LIN {X 0,Y 354.919,Z 337.275,A -85,B 0,C 180,E1 -13602.581,E2 -13602.581} C_VEL
LIN {X 0,Y 354.887,Z 337.28,A -85,B 0,C 180,E1 -13606.096,E2 -13606.096} C_VEL
LIN {X 0,Y 354.904,Z 337.277,A -85,B 0,C 180,E1 -13608.472,E2 -13608.472} C_VEL
LIN {X 0,Y 354.833,Z 337.288,A -85,B 0,C 180,E1 -13612.107,E2 -13612.107} C_VEL
LIN {X 0,Y 354.897,Z 337.277,A -85,B 0,C 180,E1 -13615.828,E2 -13615.828} C_VEL
LIN {X 0,Y 354.816,Z 337.287,A -85,B 0,C 180,E1 -13619.682,E2 -13619.682} C_VEL
LIN {X 0,Y 354.805,Z 337.288,A -85,B 0,C 180,E1 -13623.703,E2 -13623.703} C_VEL
LIN {X 0,Y 354.798,Z 337.29,A -85,B 0,C 180,E1 -13626.46,E2 -13626.46} C_VEL
LIN {X 0,Y 354.823,Z 337.285,A -85,B 0,C 180,E1 -13629.424,E2 -13629.424} C_VEL
LIN {X 0,Y 354.786,Z 337.289,A -85,B 0,C 180,E1 -13632.695,E2 -13632.695} C_VEL
LIN {X 0,Y 354.114,Z 337.376,A -85,B 0,C 180,E1 -13633.641,E2 -13633.641} C_VEL
LIN {X 0,Y 351.229,Z 337.732,A -85,B 0,C 180,E1 -13635.178,E2 -13635.178} C_VEL
LIN {X 0,Y 348.801,Z 338.036,A -85,B 0,C 180,E1 -13636.423,E2 -13636.423} C_VEL
LIN {X 0,Y 347.786,Z 338.161,A -85,B 0,C 180,E1 -13637.387,E2 -13637.387} C_VEL
LIN {X 0,Y 347.718,Z 338.169,A -85,B 0,C 180,E1 -13637.713,E2 -13637.713} C_VEL
LIN {X 0,Y 347.752,Z 338.165,A -85,B 0,C 180,E1 -13641.208,E2 -13641.208} C_VEL
LIN {X 0,Y 347.789,Z 338.164,A -85,B 0,C 180,E1 -13644.126,E2 -13644.126} C_VEL
LIN {X 0,Y 347.74,Z 338.17,A -85,B 0,C 180,E1 -13648.087,E2 -13648.087} C_VEL
LIN {X 0,Y 347.866,Z 338.151,A -85,B 0,C 180,E1 -13651.134,E2 -13651.134} C_VEL
LIN {X 0,Y 354.099,Z 357.245,A -85,B 0,C 180,E1 -13651.928,E2 -13651.928} C_VEL
LIN {X 0,Y 352.575,Z 425.531,A -85,B 0,C 180,E1 -13653.715,E2 -13653.715} C_VEL
LIN {X 0,Y 352.322,Z 438.618,A -85,B 0,C 180,E1 -13654.288,E2 -13654.288} C_VEL
LIN {X 0,Y 351.875,Z 452.101,A -85,B 0,C 180,E1 -13655.123,E2 -13655.123} C_VEL
LIN {X 0,Y 351.307,Z 464.045,A -85,B 0,C 180,E1 -13656.103,E2 -13656.103} C_VEL
LIN {X 0,Y 350.651,Z 475.904,A -85,B 0,C 180,E1 -13657.337,E2 -13657.337} C_VEL
LIN {X 0,Y 349.975,Z 486.089,A -85,B 0,C 180,E1 -13658.656,E2 -13658.656} C_VEL
LIN {X 0,Y 349.313,Z 494.652,A -85,B 0,C 180,E1 -13660,E2 -13660} C_VEL
LIN {X 0,Y 348.778,Z 502.203,A -85,B 0,C 180,E1 -13661.422,E2 -13661.422} C_VEL
LIN {X 0,Y 348.23,Z 510.285,A -85,B 0,C 180,E1 -13663.287,E2 -13663.287} C_VEL
LIN {X 0,Y 347.925,Z 515.474,A -85,B 0,C 180,E1 -13664.776,E2 -13664.776} C_VEL
LIN {X 0,Y 347.638,Z 520.436,A -85,B 0,C 180,E1 -13666.557,E2 -13666.557} C_VEL
LIN {X 0,Y 347.438,Z 524.191,A -85,B 0,C 180,E1 -13668.33,E2 -13668.33} C_VEL
LIN {X 0,Y 347.413,Z 526.086,A -85,B 0,C 180,E1 -13669.51,E2 -13669.51} C_VEL
LIN {X 0,Y 347.453,Z 527.538,A -85,B 0,C 180,E1 -13670.688,E2 -13670.688} C_VEL
LIN {X 0,Y 347.593,Z 528.701,A -85,B 0,C 180,E1 -13672.198,E2 -13672.198} C_VEL
LIN {X 0,Y 347.785,Z 529.183,A -85,B 0,C 180,E1 -13674.202,E2 -13674.202} C_VEL
LIN {X 0,Y 347.848,Z 528.865,A -85,B 0,C 180,E1 -13675.365,E2 -13675.365} C_VEL
LIN {X 0,Y 348.18,Z 528.105,A -85,B 0,C 180,E1 -13676.529,E2 -13676.529} C_VEL
LIN {X 0,Y 348.507,Z 526.945,A -85,B 0,C 180,E1 -13677.689,E2 -13677.689} C_VEL
LIN {X 0,Y 349.141,Z 524.323,A -85,B 0,C 180,E1 -13679.424,E2 -13679.424} C_VEL
LIN {X 0,Y 349.883,Z 520.636,A -85,B 0,C 180,E1 -13681.152,E2 -13681.152} C_VEL
LIN {X 0,Y 350.847,Z 515.743,A -85,B 0,C 180,E1 -13682.871,E2 -13682.871} C_VEL
LIN {X 0,Y 351.922,Z 509.602,A -85,B 0,C 180,E1 -13684.582,E2 -13684.582} C_VEL
LIN {X 0,Y 353.246,Z 501.914,A -85,B 0,C 180,E1 -13686.283,E2 -13686.283} C_VEL
LIN {X 0,Y 354.34,Z 494.044,A -85,B 0,C 180,E1 -13687.694,E2 -13687.694} C_VEL
LIN {X 0,Y 355.681,Z 484.348,A -85,B 0,C 180,E1 -13689.096,E2 -13689.096} C_VEL
LIN {X 0,Y 356.808,Z 473.673,A -85,B 0,C 180,E1 -13690.355,E2 -13690.355} C_VEL
LIN {X 0,Y 357.981,Z 461.641,A -85,B 0,C 180,E1 -13691.466,E2 -13691.466} C_VEL
LIN {X 0,Y 358.844,Z 448.971,A -85,B 0,C 180,E1 -13692.37,E2 -13692.37} C_VEL
LIN {X 0,Y 359.418,Z 435.559,A -85,B 0,C 180,E1 -13693.068,E2 -13693.068} C_VEL
LIN {X 0,Y 359.955,Z 415.445,A -85,B 0,C 180,E1 -13693.729,E2 -13693.729} C_VEL
LIN {X 0,Y 362.512,Z 365.478,A -85,B 0,C 180,E1 -13695.192,E2 -13695.192} C_VEL
LIN {X 0,Y 357.377,Z 355.182,A -85,B 0,C 180,E1 -13696.181,E2 -13696.181} C_VEL
LIN {X 0,Y 352.177,Z 346.136,A -85,B 0,C 180,E1 -13697.226,E2 -13697.226} C_VEL
LIN {X 0,Y 349.985,Z 342.457,A -85,B 0,C 180,E1 -13697.684,E2 -13697.684} C_VEL
LIN {X 0,Y 348.202,Z 339.745,A -85,B 0,C 180,E1 -13698.061,E2 -13698.061} C_VEL
LIN {X 0,Y 347.81,Z 338.162,A -85,B 0,C 180,E1 -13698.193,E2 -13698.193} C_VEL
LIN {X 0,Y 347.767,Z 338.171,A -85,B 0,C 180,E1 -13701.624,E2 -13701.624} C_VEL
LIN {X 0,Y 347.742,Z 338.171,A -85,B 0,C 180,E1 -13705.114,E2 -13705.114} C_VEL
LIN {X 0,Y 347.732,Z 338.171,A -85,B 0,C 180,E1 -13707.701,E2 -13707.701} C_VEL
LIN {X 0,Y 347.742,Z 338.169,A -85,B 0,C 180,E1 -13710.349,E2 -13710.349} C_VEL
LIN {X 0,Y 347.752,Z 338.167,A -85,B 0,C 180,E1 -13714.044,E2 -13714.044} C_VEL
LIN {X 0,Y 347.758,Z 338.163,A -85,B 0,C 180,E1 -13717.322,E2 -13717.322} C_VEL
LIN {X 0,Y 347.7,Z 338.171,A -85,B 0,C 180,E1 -13720.302,E2 -13720.302} C_VEL
LIN {X 0,Y 347.725,Z 338.169,A -85,B 0,C 180,E1 -13723.409,E2 -13723.409} C_VEL
LIN {X 0,Y 347.728,Z 338.171,A -85,B 0,C 180,E1 -13726.687,E2 -13726.687} C_VEL
LIN {X 0,Y 347.704,Z 338.174,A -85,B 0,C 180,E1 -13730.182,E2 -13730.182} C_VEL
LIN {X 0,Y 347.76,Z 338.167,A -85,B 0,C 180,E1 -13732.678,E2 -13732.678} C_VEL
LIN {X 0,Y 347.845,Z 338.187,A -85,B 0,C 180,E1 -13736.04,E2 -13736.04} C_VEL
LIN {X 0,Y 351.883,Z 357.108,A -85,B 0,C 180,E1 -13740.045,E2 -13740.045} C_VEL
LIN {X 0,Y 352.906,Z 362.731,A -85,B 0,C 180,E1 -13741.194,E2 -13741.194} C_VEL
LIN {X 0,Y 351.557,Z 377.008,A -85,B 0,C 180,E1 -13743.868,E2 -13743.868} C_VEL
LIN {X 0,Y 354.305,Z 396.014,A -85,B 0,C 180,E1 -13744.981,E2 -13744.981} C_VEL
LIN {X 0,Y 357.252,Z 419.557,A -85,B 0,C 180,E1 -13746.175,E2 -13746.175} C_VEL
LIN {X 0,Y 358.896,Z 440.791,A -85,B 0,C 180,E1 -13747.091,E2 -13747.091} C_VEL
LIN {X 0,Y 359.227,Z 450.079,A -85,B 0,C 180,E1 -13747.438,E2 -13747.438} C_VEL
LIN {X 0,Y 356.819,Z 505.004,A -85,B 0,C 180,E1 -13749.046,E2 -13749.046} C_VEL
LIN {X 0,Y 355.705,Z 518.327,A -85,B 0,C 180,E1 -13749.62,E2 -13749.62} C_VEL
LIN {X 0,Y 354.275,Z 531.746,A -85,B 0,C 180,E1 -13750.442,E2 -13750.442} C_VEL
LIN {X 0,Y 352.778,Z 543.828,A -85,B 0,C 180,E1 -13751.412,E2 -13751.412} C_VEL
LIN {X 0,Y 351.378,Z 554.869,A -85,B 0,C 180,E1 -13752.541,E2 -13752.541} C_VEL
LIN {X 0,Y 349.79,Z 566.092,A -85,B 0,C 180,E1 -13753.962,E2 -13753.962} C_VEL
LIN {X 0,Y 348.701,Z 574.974,A -85,B 0,C 180,E1 -13755.339,E2 -13755.339} C_VEL
LIN {X 0,Y 347.832,Z 583.104,A -85,B 0,C 180,E1 -13756.861,E2 -13756.861} C_VEL
LIN {X 0,Y 347.162,Z 590.742,A -85,B 0,C 180,E1 -13758.616,E2 -13758.616} C_VEL
LIN {X 0,Y 346.754,Z 597.875,A -85,B 0,C 180,E1 -13760.668,E2 -13760.668} C_VEL
LIN {X 0,Y 346.667,Z 602.629,A -85,B 0,C 180,E1 -13762.428,E2 -13762.428} C_VEL
LIN {X 0,Y 346.808,Z 606.238,A -85,B 0,C 180,E1 -13764.184,E2 -13764.184} C_VEL
LIN {X 0,Y 346.947,Z 608.034,A -85,B 0,C 180,E1 -13765.352,E2 -13765.352} C_VEL
LIN {X 0,Y 347.128,Z 610.479,A -85,B 0,C 180,E1 -13767.679,E2 -13767.679} C_VEL
LIN {X 0,Y 347.142,Z 611.524,A -85,B 0,C 180,E1 -13768.84,E2 -13768.84} C_VEL
LIN {X 0,Y 347.177,Z 612.073,A -85,B 0,C 180,E1 -13770,E2 -13770} C_VEL
LIN {X 0,Y 347.063,Z 612.157,A -85,B 0,C 180,E1 -13771.16,E2 -13771.16} C_VEL
LIN {X 0,Y 347.002,Z 611.804,A -85,B 0,C 180,E1 -13772.321,E2 -13772.321} C_VEL
LIN {X 0,Y 346.991,Z 610.97,A -85,B 0,C 180,E1 -13773.483,E2 -13773.483} C_VEL
LIN {X 0,Y 346.815,Z 609.662,A -85,B 0,C 180,E1 -13774.649,E2 -13774.649} C_VEL
LIN {X 0,Y 346.646,Z 606.55,A -85,B 0,C 180,E1 -13776.563,E2 -13776.563} C_VEL
LIN {X 0,Y 346.604,Z 602.992,A -85,B 0,C 180,E1 -13778.16,E2 -13778.16} C_VEL
LIN {X 0,Y 346.747,Z 597.974,A -85,B 0,C 180,E1 -13779.92,E2 -13779.92} C_VEL
LIN {X 0,Y 347.369,Z 590.58,A -85,B 0,C 180,E1 -13781.969,E2 -13781.969} C_VEL
LIN {X 0,Y 348.248,Z 582.607,A -85,B 0,C 180,E1 -13783.717,E2 -13783.717} C_VEL
LIN {X 0,Y 349.166,Z 574.644,A -85,B 0,C 180,E1 -13785.169,E2 -13785.169} C_VEL
LIN {X 0,Y 350.603,Z 564.098,A -85,B 0,C 180,E1 -13786.747,E2 -13786.747} C_VEL
LIN {X 0,Y 352.178,Z 553.666,A -85,B 0,C 180,E1 -13788.018,E2 -13788.018} C_VEL
LIN {X 0,Y 353.974,Z 540.75,A -85,B 0,C 180,E1 -13789.274,E2 -13789.274} C_VEL
LIN {X 0,Y 355.614,Z 528.179,A -85,B 0,C 180,E1 -13790.234,E2 -13790.234} C_VEL
LIN {X 0,Y 357.176,Z 513.944,A -85,B 0,C 180,E1 -13791.045,E2 -13791.045} C_VEL
LIN {X 0,Y 358.179,Z 500.972,A -85,B 0,C 180,E1 -13791.586,E2 -13791.586} C_VEL
LIN {X 0,Y 360.904,Z 446.729,A -85,B 0,C 180,E1 -13793.232,E2 -13793.232} C_VEL
LIN {X 0,Y 359.98,Z 429.272,A -85,B 0,C 180,E1 -13793.989,E2 -13793.989} C_VEL
LIN {X 0,Y 358.57,Z 415.657,A -85,B 0,C 180,E1 -13794.686,E2 -13794.686} C_VEL
LIN {X 0,Y 355.618,Z 397.209,A -85,B 0,C 180,E1 -13795.818,E2 -13795.818} C_VEL
LIN {X 0,Y 353.506,Z 386.369,A -85,B 0,C 180,E1 -13796.582,E2 -13796.582} C_VEL
LIN {X 0,Y 356.108,Z 371.321,A -85,B 0,C 180,E1 -13799.888,E2 -13799.888} C_VEL
LIN {X 0,Y 355.734,Z 367.471,A -85,B 0,C 180,E1 -13800.908,E2 -13800.908} C_VEL
LIN {X 0,Y 353.94,Z 358.853,A -85,B 0,C 180,E1 -13803.49,E2 -13803.49} C_VEL
LIN {X 0,Y 351.998,Z 351.5,A -85,B 0,C 180,E1 -13806.063,E2 -13806.063} C_VEL
LIN {X 0,Y 350.159,Z 345.665,A -85,B 0,C 180,E1 -13808.485,E2 -13808.485} C_VEL
LIN {X 0,Y 348.768,Z 341.487,A -85,B 0,C 180,E1 -13810.536,E2 -13810.536} C_VEL
LIN {X 0,Y 347.741,Z 338.171,A -85,B 0,C 180,E1 -13812.515,E2 -13812.515} C_VEL
LIN {X 0,Y 347.726,Z 338.172,A -85,B 0,C 180,E1 -13816.686,E2 -13816.686} C_VEL
LIN {X 0,Y 347.703,Z 338.174,A -85,B 0,C 180,E1 -13820.182,E2 -13820.182} C_VEL
LIN {X 0,Y 347.756,Z 338.166,A -85,B 0,C 180,E1 -13822.678,E2 -13822.678} C_VEL
LIN {X 0,Y 347.75,Z 338.168,A -85,B 0,C 180,E1 -13825.956,E2 -13825.956} C_VEL
LIN {X 0,Y 347.74,Z 338.17,A -85,B 0,C 180,E1 -13829.651,E2 -13829.651} C_VEL
LIN {X 0,Y 347.736,Z 338.172,A -85,B 0,C 180,E1 -13833.599,E2 -13833.599} C_VEL
LIN {X 0,Y 347.75,Z 338.251,A -85,B 0,C 180,E1 -13834.726,E2 -13834.726} C_VEL
LIN {X 0,Y 348.787,Z 341.047,A -85,B 0,C 180,E1 -13835.059,E2 -13835.059} C_VEL
LIN {X 0,Y 350.812,Z 343.515,A -85,B 0,C 180,E1 -13835.536,E2 -13835.536} C_VEL
LIN {X 0,Y 352.889,Z 346.829,A -85,B 0,C 180,E1 -13836.04,E2 -13836.04} C_VEL
LIN {X 0,Y 358.301,Z 356.024,A -85,B 0,C 180,E1 -13837.289,E2 -13837.289} C_VEL
LIN {X 0,Y 363.207,Z 365.361,A -85,B 0,C 180,E1 -13838.35,E2 -13838.35} C_VEL
LIN {X 0,Y 364.094,Z 367.357,A -85,B 0,C 180,E1 -13838.546,E2 -13838.546} C_VEL
LIN {X 0,Y 360.695,Z 423.977,A -85,B 0,C 180,E1 -13840.325,E2 -13840.325} C_VEL
LIN {X 0,Y 360.228,Z 439.497,A -85,B 0,C 180,E1 -13840.925,E2 -13840.925} C_VEL
LIN {X 0,Y 359.511,Z 452.969,A -85,B 0,C 180,E1 -13841.699,E2 -13841.699} C_VEL
LIN {X 0,Y 358.551,Z 464.924,A -85,B 0,C 180,E1 -13842.607,E2 -13842.607} C_VEL
LIN {X 0,Y 357.214,Z 477.672,A -85,B 0,C 180,E1 -13843.864,E2 -13843.864} C_VEL
LIN {X 0,Y 355.936,Z 487.766,A -85,B 0,C 180,E1 -13845.126,E2 -13845.126} C_VEL
LIN {X 0,Y 354.623,Z 496.83,A -85,B 0,C 180,E1 -13846.521,E2 -13846.521} C_VEL
LIN {X 0,Y 353.388,Z 504.455,A -85,B 0,C 180,E1 -13847.946,E2 -13847.946} C_VEL
LIN {X 0,Y 352.096,Z 511.82,A -85,B 0,C 180,E1 -13849.65,E2 -13849.65} C_VEL
LIN {X 0,Y 350.975,Z 517.659,A -85,B 0,C 180,E1 -13851.362,E2 -13851.362} C_VEL
LIN {X 0,Y 349.954,Z 522.243,A -85,B 0,C 180,E1 -13853.079,E2 -13853.079} C_VEL
LIN {X 0,Y 349.436,Z 524.653,A -85,B 0,C 180,E1 -13854.228,E2 -13854.228} C_VEL
LIN {X 0,Y 348.938,Z 526.601,A -85,B 0,C 180,E1 -13855.378,E2 -13855.378} C_VEL
LIN {X 0,Y 348.543,Z 528.056,A -85,B 0,C 180,E1 -13856.531,E2 -13856.531} C_VEL
LIN {X 0,Y 348.283,Z 529.081,A -85,B 0,C 180,E1 -13857.686,E2 -13857.686} C_VEL
LIN {X 0,Y 348.009,Z 529.697,A -85,B 0,C 180,E1 -13858.842,E2 -13858.842} C_VEL
LIN {X 0,Y 347.876,Z 529.838,A -85,B 0,C 180,E1 -13859.999,E2 -13859.999} C_VEL
LIN {X 0,Y 347.629,Z 529.59,A -85,B 0,C 180,E1 -13861.158,E2 -13861.158} C_VEL
LIN {X 0,Y 347.266,Z 528.951,A -85,B 0,C 180,E1 -13862.319,E2 -13862.319} C_VEL
LIN {X 0,Y 347.311,Z 527.804,A -85,B 0,C 180,E1 -13863.48,E2 -13863.48} C_VEL
LIN {X 0,Y 347.491,Z 526.22,A -85,B 0,C 180,E1 -13864.64,E2 -13864.64} C_VEL
LIN {X 0,Y 347.641,Z 523.023,A -85,B 0,C 180,E1 -13866.383,E2 -13866.383} C_VEL
LIN {X 0,Y 347.718,Z 518.732,A -85,B 0,C 180,E1 -13868.133,E2 -13868.133} C_VEL
LIN {X 0,Y 348.04,Z 513.213,A -85,B 0,C 180,E1 -13869.883,E2 -13869.883} C_VEL
LIN {X 0,Y 348.453,Z 506.273,A -85,B 0,C 180,E1 -13871.635,E2 -13871.635} C_VEL
LIN {X 0,Y 349.056,Z 497.611,A -85,B 0,C 180,E1 -13873.387,E2 -13873.387} C_VEL
LIN {X 0,Y 349.586,Z 488.775,A -85,B 0,C 180,E1 -13874.851,E2 -13874.851} C_VEL
LIN {X 0,Y 350.247,Z 477.885,A -85,B 0,C 180,E1 -13876.315,E2 -13876.315} C_VEL
LIN {X 0,Y 350.948,Z 465.66,A -85,B 0,C 180,E1 -13877.631,E2 -13877.631} C_VEL
LIN {X 0,Y 351.503,Z 453.438,A -85,B 0,C 180,E1 -13878.657,E2 -13878.657} C_VEL
LIN {X 0,Y 352.064,Z 441.042,A -85,B 0,C 180,E1 -13879.458,E2 -13879.458} C_VEL
LIN {X 0,Y 352.342,Z 427.98,A -85,B 0,C 180,E1 -13880.073,E2 -13880.073} C_VEL
LIN {X 0,Y 352.569,Z 409.14,A -85,B 0,C 180,E1 -13880.634,E2 -13880.634} C_VEL
LIN {X 0,Y 353.835,Z 357.031,A -85,B 0,C 180,E1 -13882.025,E2 -13882.025} C_VEL
LIN {X 0,Y 347.808,Z 338.163,A -85,B 0,C 180,E1 -13882.812,E2 -13882.812} C_VEL
LIN {X 0,Y 347.832,Z 338.156,A -85,B 0,C 180,E1 -13886.392,E2 -13886.392} C_VEL
LIN {X 0,Y 347.808,Z 338.158,A -85,B 0,C 180,E1 -13889.671,E2 -13889.671} C_VEL
LIN {X 0,Y 347.732,Z 338.171,A -85,B 0,C 180,E1 -13893.071,E2 -13893.071} C_VEL
LIN {X 0,Y 347.769,Z 338.163,A -85,B 0,C 180,E1 -13896.064,E2 -13896.064} C_VEL
LIN {X 0,Y 347.75,Z 338.17,A -85,B 0,C 180,E1 -13898.792,E2 -13898.792} C_VEL
LIN {X 0,Y 347.749,Z 338.165,A -85,B 0,C 180,E1 -13901.83,E2 -13901.83} C_VEL
LIN {X 0,Y 347.763,Z 338.166,A -85,B 0,C 180,E1 -13905.016,E2 -13905.016} C_VEL
LIN {X 0,Y 347.748,Z 338.168,A -85,B 0,C 180,E1 -13908.397,E2 -13908.397} C_VEL
LIN {X 0,Y 347.775,Z 338.162,A -85,B 0,C 180,E1 -13912.01,E2 -13912.01} C_VEL
LIN {X 0,Y 347.742,Z 338.166,A -85,B 0,C 180,E1 -13915.536,E2 -13915.536} C_VEL
LIN {X 0,Y 347.742,Z 338.169,A -85,B 0,C 180,E1 -13918.3,E2 -13918.3} C_VEL
LIN {X 0,Y 347.776,Z 338.164,A -85,B 0,C 180,E1 -13920.987,E2 -13920.987} C_VEL
LIN {X 0,Y 347.828,Z 338.155,A -85,B 0,C 180,E1 -13923.607,E2 -13923.607} C_VEL
LIN {X 0,Y 347.786,Z 338.162,A -85,B 0,C 180,E1 -13926.162,E2 -13926.162} C_VEL
LIN {X 0,Y 347.81,Z 338.158,A -85,B 0,C 180,E1 -13929.909,E2 -13929.909} C_VEL
LIN {X 0,Y 347.863,Z 338.155,A -85,B 0,C 180,E1 -13932.359,E2 -13932.359} C_VEL
LIN {X 0,Y 347.894,Z 338.148,A -85,B 0,C 180,E1 -13935.971,E2 -13935.971} C_VEL
LIN {X 0,Y 347.927,Z 338.143,A -85,B 0,C 180,E1 -13939.526,E2 -13939.526} C_VEL
LIN {X 0,Y 348.072,Z 338.126,A -85,B 0,C 180,E1 -13941.875,E2 -13941.875} C_VEL
LIN {X 0,Y 348.065,Z 338.129,A -85,B 0,C 180,E1 -13944.206,E2 -13944.206} C_VEL
LIN {X 0,Y 348.206,Z 338.109,A -85,B 0,C 180,E1 -13947.687,E2 -13947.687} C_VEL
LIN {X 0,Y 348.344,Z 338.093,A -85,B 0,C 180,E1 -13950,E2 -13950} C_VEL
LIN {X 0,Y 348.206,Z 338.114,A -85,B 0,C 180,E1 -13952.314,E2 -13952.314} C_VEL
LIN {X 0,Y 348.104,Z 338.122,A -85,B 0,C 180,E1 -13956.958,E2 -13956.958} C_VEL
LIN {X 0,Y 347.965,Z 338.138,A -85,B 0,C 180,E1 -13959.299,E2 -13959.299} C_VEL
LIN {X 0,Y 347.888,Z 338.149,A -85,B 0,C 180,E1 -13962.84,E2 -13962.84} C_VEL
LIN {X 0,Y 347.837,Z 338.158,A -85,B 0,C 180,E1 -13966.432,E2 -13966.432} C_VEL
LIN {X 0,Y 347.854,Z 338.153,A -85,B 0,C 180,E1 -13968.861,E2 -13968.861} C_VEL
LIN {X 0,Y 347.772,Z 338.165,A -85,B 0,C 180,E1 -13972.58,E2 -13972.58} C_VEL
LIN {X 0,Y 347.81,Z 338.157,A -85,B 0,C 180,E1 -13975.109,E2 -13975.109} C_VEL
LIN {X 0,Y 347.806,Z 338.16,A -85,B 0,C 180,E1 -13977.695,E2 -13977.695} C_VEL
LIN {X 0,Y 347.747,Z 338.169,A -85,B 0,C 180,E1 -13980.349,E2 -13980.349} C_VEL
LIN {X 0,Y 347.747,Z 338.171,A -85,B 0,C 180,E1 -13984.044,E2 -13984.044} C_VEL
LIN {X 0,Y 347.762,Z 338.164,A -85,B 0,C 180,E1 -13987.321,E2 -13987.321} C_VEL
LIN {X 0,Y 347.732,Z 338.171,A -85,B 0,C 180,E1 -13990.298,E2 -13990.298} C_VEL
LIN {X 0,Y 347.723,Z 338.169,A -85,B 0,C 180,E1 -13993.409,E2 -13993.409} C_VEL
LIN {X 0,Y 347.725,Z 338.169,A -85,B 0,C 180,E1 -13996.687,E2 -13996.687} C_VEL
LIN {X 0,Y 347.718,Z 338.169,A -85,B 0,C 180,E1 -13997.713,E2 -13997.713} C_VEL
LIN {X 0,Y 347.086,Z 338.252,A -85,B 0,C 180,E1 -13998.679,E2 -13998.679} C_VEL
LIN {X 0,Y 344.233,Z 338.607,A -85,B 0,C 180,E1 -14000.25,E2 -14000.25} C_VEL
LIN {X 0,Y 341.802,Z 338.908,A -85,B 0,C 180,E1 -14001.523,E2 -14001.523} C_VEL
LIN {X 0,Y 340.767,Z 339.036,A -85,B 0,C 180,E1 -14002.507,E2 -14002.507} C_VEL
LIN {X 0,Y 340.69,Z 339.043,A -85,B 0,C 180,E1 -14002.841,E2 -14002.841} C_VEL
LIN {X 0,Y 340.693,Z 339.048,A -85,B 0,C 180,E1 -14006.154,E2 -14006.154} C_VEL
LIN {X 0,Y 340.792,Z 339.032,A -85,B 0,C 180,E1 -14010.595,E2 -14010.595} C_VEL
LIN {X 0,Y 340.821,Z 339.028,A -85,B 0,C 180,E1 -14010.833,E2 -14010.833} C_VEL
LIN {X 0,Y 347.167,Z 358.525,A -85,B 0,C 180,E1 -14011.679,E2 -14011.679} C_VEL
LIN {X 0,Y 345.608,Z 426.565,A -85,B 0,C 180,E1 -14013.514,E2 -14013.514} C_VEL
LIN {X 0,Y 345.367,Z 438.782,A -85,B 0,C 180,E1 -14014.055,E2 -14014.055} C_VEL
LIN {X 0,Y 344.924,Z 452.416,A -85,B 0,C 180,E1 -14014.909,E2 -14014.909} C_VEL
LIN {X 0,Y 344.322,Z 464.495,A -85,B 0,C 180,E1 -14015.907,E2 -14015.907} C_VEL
LIN {X 0,Y 343.658,Z 476.165,A -85,B 0,C 180,E1 -14017.136,E2 -14017.136} C_VEL
LIN {X 0,Y 342.957,Z 486.706,A -85,B 0,C 180,E1 -14018.513,E2 -14018.513} C_VEL
LIN {X 0,Y 342.172,Z 497.057,A -85,B 0,C 180,E1 -14020.191,E2 -14020.191} C_VEL
LIN {X 0,Y 341.597,Z 504.989,A -85,B 0,C 180,E1 -14021.774,E2 -14021.774} C_VEL
LIN {X 0,Y 341.111,Z 512.158,A -85,B 0,C 180,E1 -14023.544,E2 -14023.544} C_VEL
LIN {X 0,Y 340.7,Z 518.94,A -85,B 0,C 180,E1 -14025.669,E2 -14025.669} C_VEL
LIN {X 0,Y 340.498,Z 523.302,A -85,B 0,C 180,E1 -14027.484,E2 -14027.484} C_VEL
LIN {X 0,Y 340.365,Z 526.528,A -85,B 0,C 180,E1 -14029.291,E2 -14029.291} C_VEL
LIN {X 0,Y 340.399,Z 528.087,A -85,B 0,C 180,E1 -14030.493,E2 -14030.493} C_VEL
LIN {X 0,Y 340.548,Z 529.497,A -85,B 0,C 180,E1 -14032.138,E2 -14032.138} C_VEL
LIN {X 0,Y 340.736,Z 530.124,A -85,B 0,C 180,E1 -14034.081,E2 -14034.081} C_VEL
LIN {X 0,Y 340.819,Z 529.973,A -85,B 0,C 180,E1 -14035.269,E2 -14035.269} C_VEL
LIN {X 0,Y 341.159,Z 529.314,A -85,B 0,C 180,E1 -14036.457,E2 -14036.457} C_VEL
LIN {X 0,Y 341.492,Z 528.252,A -85,B 0,C 180,E1 -14037.642,E2 -14037.642} C_VEL
LIN {X 0,Y 341.931,Z 526.761,A -85,B 0,C 180,E1 -14038.823,E2 -14038.823} C_VEL
LIN {X 0,Y 342.67,Z 523.656,A -85,B 0,C 180,E1 -14040.588,E2 -14040.588} C_VEL
LIN {X 0,Y 343.589,Z 519.435,A -85,B 0,C 180,E1 -14042.345,E2 -14042.345} C_VEL
LIN {X 0,Y 344.866,Z 512.946,A -85,B 0,C 180,E1 -14044.383,E2 -14044.383} C_VEL
LIN {X 0,Y 346.189,Z 505.817,A -85,B 0,C 180,E1 -14046.119,E2 -14046.119} C_VEL
LIN {X 0,Y 347.628,Z 496.879,A -85,B 0,C 180,E1 -14047.844,E2 -14047.844} C_VEL
LIN {X 0,Y 348.997,Z 487.751,A -85,B 0,C 180,E1 -14049.271,E2 -14049.271} C_VEL
LIN {X 0,Y 350.415,Z 476.366,A -85,B 0,C 180,E1 -14050.692,E2 -14050.692} C_VEL
LIN {X 0,Y 351.493,Z 466.447,A -85,B 0,C 180,E1 -14051.681,E2 -14051.681} C_VEL
LIN {X 0,Y 352.542,Z 453.809,A -85,B 0,C 180,E1 -14052.668,E2 -14052.668} C_VEL
LIN {X 0,Y 353.177,Z 441.312,A -85,B 0,C 180,E1 -14053.413,E2 -14053.413} C_VEL
LIN {X 0,Y 353.643,Z 427.38,A -85,B 0,C 180,E1 -14053.981,E2 -14053.981} C_VEL
LIN {X 0,Y 355.261,Z 393.299,A -85,B 0,C 180,E1 -14055.013,E2 -14055.013} C_VEL
LIN {X 0,Y 356.575,Z 367.631,A -85,B 0,C 180,E1 -14055.807,E2 -14055.807} C_VEL
LIN {X 0,Y 350.956,Z 356.567,A -85,B 0,C 180,E1 -14056.97,E2 -14056.97} C_VEL
LIN {X 0,Y 345.465,Z 347.324,A -85,B 0,C 180,E1 -14058.144,E2 -14058.144} C_VEL
LIN {X 0,Y 343.016,Z 343.428,A -85,B 0,C 180,E1 -14058.701,E2 -14058.701} C_VEL
LIN {X 0,Y 341.215,Z 340.927,A -85,B 0,C 180,E1 -14059.104,E2 -14059.104} C_VEL
LIN {X 0,Y 340.706,Z 339.051,A -85,B 0,C 180,E1 -14059.272,E2 -14059.272} C_VEL
LIN {X 0,Y 340.704,Z 339.044,A -85,B 0,C 180,E1 -14063.075,E2 -14063.075} C_VEL
LIN {X 0,Y 340.714,Z 339.046,A -85,B 0,C 180,E1 -14066.988,E2 -14066.988} C_VEL
LIN {X 0,Y 340.697,Z 339.047,A -85,B 0,C 180,E1 -14071.045,E2 -14071.045} C_VEL
LIN {X 0,Y 340.719,Z 339.039,A -85,B 0,C 180,E1 -14075.279,E2 -14075.279} C_VEL
LIN {X 0,Y 340.697,Z 339.042,A -85,B 0,C 180,E1 -14078.382,E2 -14078.382} C_VEL
LIN {X 0,Y 340.695,Z 339.044,A -85,B 0,C 180,E1 -14082.044,E2 -14082.044} C_VEL
LIN {X 0,Y 340.654,Z 339.053,A -85,B 0,C 180,E1 -14086.227,E2 -14086.227} C_VEL
LIN {X 0,Y 340.674,Z 339.048,A -85,B 0,C 180,E1 -14088.688,E2 -14088.688} C_VEL
LIN {X 0,Y 340.723,Z 339.044,A -85,B 0,C 180,E1 -14091.771,E2 -14091.771} C_VEL
LIN {X 0,Y 340.792,Z 339.058,A -85,B 0,C 180,E1 -14095.788,E2 -14095.788} C_VEL
LIN {X 0,Y 344.662,Z 357.079,A -85,B 0,C 180,E1 -14099.69,E2 -14099.69} C_VEL
LIN {X 0,Y 345.917,Z 363.68,A -85,B 0,C 180,E1 -14101.067,E2 -14101.067} C_VEL
LIN {X 0,Y 345.06,Z 372.098,A -85,B 0,C 180,E1 -14102.677,E2 -14102.677} C_VEL
LIN {X 0,Y 345.866,Z 378.841,A -85,B 0,C 180,E1 -14103.203,E2 -14103.203} C_VEL
LIN {X 0,Y 348.728,Z 398.321,A -85,B 0,C 180,E1 -14104.374,E2 -14104.374} C_VEL
LIN {X 0,Y 351.476,Z 421.811,A -85,B 0,C 180,E1 -14105.614,E2 -14105.614} C_VEL
LIN {X 0,Y 352.911,Z 442.461,A -85,B 0,C 180,E1 -14106.528,E2 -14106.528} C_VEL
LIN {X 0,Y 353.174,Z 450.553,A -85,B 0,C 180,E1 -14106.847,E2 -14106.847} C_VEL
LIN {X 0,Y 350.637,Z 504.238,A -85,B 0,C 180,E1 -14108.466,E2 -14108.466} C_VEL
LIN {X 0,Y 349.422,Z 517.92,A -85,B 0,C 180,E1 -14109.083,E2 -14109.083} C_VEL
LIN {X 0,Y 347.903,Z 531.016,A -85,B 0,C 180,E1 -14109.914,E2 -14109.914} C_VEL
LIN {X 0,Y 346.283,Z 542.969,A -85,B 0,C 180,E1 -14110.897,E2 -14110.897} C_VEL
LIN {X 0,Y 344.809,Z 553.97,A -85,B 0,C 180,E1 -14112.044,E2 -14112.044} C_VEL
LIN {X 0,Y 343.117,Z 565.171,A -85,B 0,C 180,E1 -14113.489,E2 -14113.489} C_VEL
LIN {X 0,Y 341.963,Z 573.703,A -85,B 0,C 180,E1 -14114.841,E2 -14114.841} C_VEL
LIN {X 0,Y 340.887,Z 582.765,A -85,B 0,C 180,E1 -14116.588,E2 -14116.588} C_VEL
LIN {X 0,Y 340.156,Z 590.303,A -85,B 0,C 180,E1 -14118.378,E2 -14118.378} C_VEL
LIN {X 0,Y 339.697,Z 597.33,A -85,B 0,C 180,E1 -14120.473,E2 -14120.473} C_VEL
LIN {X 0,Y 339.574,Z 601.968,A -85,B 0,C 180,E1 -14122.268,E2 -14122.268} C_VEL
LIN {X 0,Y 339.717,Z 605.503,A -85,B 0,C 180,E1 -14124.063,E2 -14124.063} C_VEL
LIN {X 0,Y 339.851,Z 607.244,A -85,B 0,C 180,E1 -14125.255,E2 -14125.255} C_VEL
LIN {X 0,Y 340.01,Z 608.552,A -85,B 0,C 180,E1 -14126.445,E2 -14126.445} C_VEL
LIN {X 0,Y 340.114,Z 610.46,A -85,B 0,C 180,E1 -14128.816,E2 -14128.816} C_VEL
LIN {X 0,Y 340.145,Z 611.078,A -85,B 0,C 180,E1 -14130,E2 -14130} C_VEL
LIN {X 0,Y 340.023,Z 611.202,A -85,B 0,C 180,E1 -14131.184,E2 -14131.184} C_VEL
LIN {X 0,Y 339.952,Z 610.888,A -85,B 0,C 180,E1 -14132.369,E2 -14132.369} C_VEL
LIN {X 0,Y 339.914,Z 610.132,A -85,B 0,C 180,E1 -14133.556,E2 -14133.556} C_VEL
LIN {X 0,Y 339.726,Z 608.866,A -85,B 0,C 180,E1 -14134.746,E2 -14134.746} C_VEL
LIN {X 0,Y 339.578,Z 606.084,A -85,B 0,C 180,E1 -14136.572,E2 -14136.572} C_VEL
LIN {X 0,Y 339.534,Z 602.373,A -85,B 0,C 180,E1 -14138.331,E2 -14138.331} C_VEL
LIN {X 0,Y 339.687,Z 597.465,A -85,B 0,C 180,E1 -14140.129,E2 -14140.129} C_VEL
LIN {X 0,Y 340.352,Z 590.187,A -85,B 0,C 180,E1 -14142.219,E2 -14142.219} C_VEL
LIN {X 0,Y 341.323,Z 582.418,A -85,B 0,C 180,E1 -14144.001,E2 -14144.001} C_VEL
LIN {X 0,Y 342.295,Z 574.634,A -85,B 0,C 180,E1 -14145.481,E2 -14145.481} C_VEL
LIN {X 0,Y 343.814,Z 564.309,A -85,B 0,C 180,E1 -14147.088,E2 -14147.088} C_VEL
LIN {X 0,Y 345.66,Z 552.942,A -85,B 0,C 180,E1 -14148.523,E2 -14148.523} C_VEL
LIN {X 0,Y 347.556,Z 540.196,A -85,B 0,C 180,E1 -14149.798,E2 -14149.798} C_VEL
LIN {X 0,Y 349.304,Z 527.861,A -85,B 0,C 180,E1 -14150.77,E2 -14150.77} C_VEL
LIN {X 0,Y 350.933,Z 514.069,A -85,B 0,C 180,E1 -14151.592,E2 -14151.592} C_VEL
LIN {X 0,Y 352.15,Z 499.983,A -85,B 0,C 180,E1 -14152.206,E2 -14152.206} C_VEL
LIN {X 0,Y 355.024,Z 447.812,A -85,B 0,C 180,E1 -14153.842,E2 -14153.842} C_VEL
LIN {X 0,Y 354.244,Z 430.974,A -85,B 0,C 180,E1 -14154.6,E2 -14154.6} C_VEL
LIN {X 0,Y 352.912,Z 417.083,A -85,B 0,C 180,E1 -14155.339,E2 -14155.339} C_VEL
LIN {X 0,Y 349.914,Z 397.616,A -85,B 0,C 180,E1 -14156.596,E2 -14156.596} C_VEL
LIN {X 0,Y 347.354,Z 384.705,A -85,B 0,C 180,E1 -14157.596,E2 -14157.596} C_VEL
LIN {X 0,Y 349.525,Z 373.297,A -85,B 0,C 180,E1 -14160.178,E2 -14160.178} C_VEL
LIN {X 0,Y 348.91,Z 368.295,A -85,B 0,C 180,E1 -14161.582,E2 -14161.582} C_VEL
LIN {X 0,Y 347.306,Z 360.878,A -85,B 0,C 180,E1 -14163.935,E2 -14163.935} C_VEL
LIN {X 0,Y 345.754,Z 354.831,A -85,B 0,C 180,E1 -14166.12,E2 -14166.12} C_VEL
LIN {X 0,Y 343.435,Z 347.412,A -85,B 0,C 180,E1 -14169.374,E2 -14169.374} C_VEL
LIN {X 0,Y 341.722,Z 342.262,A -85,B 0,C 180,E1 -14172.234,E2 -14172.234} C_VEL
LIN {X 0,Y 340.65,Z 339.054,A -85,B 0,C 180,E1 -14174.544,E2 -14174.544} C_VEL
LIN {X 0,Y 340.695,Z 339.048,A -85,B 0,C 180,E1 -14177.955,E2 -14177.955} C_VEL
LIN {X 0,Y 340.72,Z 339.042,A -85,B 0,C 180,E1 -14181.77,E2 -14181.77} C_VEL
LIN {X 0,Y 340.724,Z 339.042,A -85,B 0,C 180,E1 -14185.595,E2 -14185.595} C_VEL
LIN {X 0,Y 340.695,Z 339.048,A -85,B 0,C 180,E1 -14188.954,E2 -14188.954} C_VEL
LIN {X 0,Y 340.712,Z 339.046,A -85,B 0,C 180,E1 -14193.011,E2 -14193.011} C_VEL
LIN {X 0,Y 340.708,Z 339.166,A -85,B 0,C 180,E1 -14193.397,E2 -14193.397} C_VEL
LIN {X 0,Y 341.716,Z 341.936,A -85,B 0,C 180,E1 -14193.762,E2 -14193.762} C_VEL
LIN {X 0,Y 343.861,Z 344.302,A -85,B 0,C 180,E1 -14194.32,E2 -14194.32} C_VEL
LIN {X 0,Y 345.791,Z 347.633,A -85,B 0,C 180,E1 -14194.862,E2 -14194.862} C_VEL
LIN {X 0,Y 347.068,Z 349.378,A -85,B 0,C 180,E1 -14195.183,E2 -14195.183} C_VEL
LIN {X 0,Y 352.117,Z 357.784,A -85,B 0,C 180,E1 -14196.441,E2 -14196.441} C_VEL
LIN {X 0,Y 357.119,Z 367.115,A -85,B 0,C 180,E1 -14197.606,E2 -14197.606} C_VEL
LIN {X 0,Y 358.453,Z 370.29,A -85,B 0,C 180,E1 -14197.928,E2 -14197.928} C_VEL
LIN {X 0,Y 354.909,Z 423.481,A -85,B 0,C 180,E1 -14199.648,E2 -14199.648} C_VEL
LIN {X 0,Y 354.364,Z 440.009,A -85,B 0,C 180,E1 -14200.296,E2 -14200.296} C_VEL
LIN {X 0,Y 353.641,Z 452.467,A -85,B 0,C 180,E1 -14201.008,E2 -14201.008} C_VEL
LIN {X 0,Y 352.537,Z 465.573,A -85,B 0,C 180,E1 -14202,E2 -14202} C_VEL
LIN {X 0,Y 351.101,Z 478.331,A -85,B 0,C 180,E1 -14203.276,E2 -14203.276} C_VEL
LIN {X 0,Y 349.749,Z 488.487,A -85,B 0,C 180,E1 -14204.558,E2 -14204.558} C_VEL
LIN {X 0,Y 348.115,Z 498.89,A -85,B 0,C 180,E1 -14206.2,E2 -14206.2} C_VEL
LIN {X 0,Y 346.752,Z 506.612,A -85,B 0,C 180,E1 -14207.712,E2 -14207.712} C_VEL
LIN {X 0,Y 345.342,Z 513.711,A -85,B 0,C 180,E1 -14209.446,E2 -14209.446} C_VEL
LIN {X 0,Y 344.151,Z 519.376,A -85,B 0,C 180,E1 -14211.189,E2 -14211.189} C_VEL
LIN {X 0,Y 343.091,Z 523.789,A -85,B 0,C 180,E1 -14212.94,E2 -14212.94} C_VEL
LIN {X 0,Y 342.532,Z 526.115,A -85,B 0,C 180,E1 -14214.111,E2 -14214.111} C_VEL
LIN {X 0,Y 342.01,Z 527.929,A -85,B 0,C 180,E1 -14215.285,E2 -14215.285} C_VEL
LIN {X 0,Y 341.573,Z 529.31,A -85,B 0,C 180,E1 -14216.461,E2 -14216.461} C_VEL
LIN {X 0,Y 341.297,Z 530.253,A -85,B 0,C 180,E1 -14217.639,E2 -14217.639} C_VEL
LIN {X 0,Y 340.99,Z 530.749,A -85,B 0,C 180,E1 -14218.818,E2 -14218.818} C_VEL
LIN {X 0,Y 340.854,Z 530.81,A -85,B 0,C 180,E1 -14219.999,E2 -14219.999} C_VEL
LIN {X 0,Y 340.593,Z 530.487,A -85,B 0,C 180,E1 -14221.182,E2 -14221.182} C_VEL
LIN {X 0,Y 340.214,Z 529.732,A -85,B 0,C 180,E1 -14222.367,E2 -14222.367} C_VEL
LIN {X 0,Y 340.274,Z 528.49,A -85,B 0,C 180,E1 -14223.552,E2 -14223.552} C_VEL
LIN {X 0,Y 340.503,Z 525.819,A -85,B 0,C 180,E1 -14225.329,E2 -14225.329} C_VEL
LIN {X 0,Y 340.58,Z 521.882,A -85,B 0,C 180,E1 -14227.207,E2 -14227.207} C_VEL
LIN {X 0,Y 340.827,Z 517.25,A -85,B 0,C 180,E1 -14228.896,E2 -14228.896} C_VEL
LIN {X 0,Y 341.164,Z 511.095,A -85,B 0,C 180,E1 -14230.684,E2 -14230.684} C_VEL
LIN {X 0,Y 341.643,Z 503.382,A -85,B 0,C 180,E1 -14232.473,E2 -14232.473} C_VEL
LIN {X 0,Y 342.308,Z 493.783,A -85,B 0,C 180,E1 -14234.262,E2 -14234.262} C_VEL
LIN {X 0,Y 342.891,Z 483.856,A -85,B 0,C 180,E1 -14235.757,E2 -14235.757} C_VEL
LIN {X 0,Y 343.596,Z 472.859,A -85,B 0,C 180,E1 -14237.099,E2 -14237.099} C_VEL
LIN {X 0,Y 344.225,Z 460.628,A -85,B 0,C 180,E1 -14238.294,E2 -14238.294} C_VEL
LIN {X 0,Y 344.863,Z 447.809,A -85,B 0,C 180,E1 -14239.261,E2 -14239.261} C_VEL
LIN {X 0,Y 345.262,Z 434.473,A -85,B 0,C 180,E1 -14240.012,E2 -14240.012} C_VEL
LIN {X 0,Y 345.433,Z 420.247,A -85,B 0,C 180,E1 -14240.552,E2 -14240.552} C_VEL
LIN {X 0,Y 346.856,Z 358.067,A -85,B 0,C 180,E1 -14242.269,E2 -14242.269} C_VEL
LIN {X 0,Y 340.783,Z 339.037,A -85,B 0,C 180,E1 -14243.088,E2 -14243.088} C_VEL
LIN {X 0,Y 340.804,Z 339.035,A -85,B 0,C 180,E1 -14246.979,E2 -14246.979} C_VEL
LIN {X 0,Y 340.763,Z 339.035,A -85,B 0,C 180,E1 -14249.977,E2 -14249.977} C_VEL
LIN {X 0,Y 340.691,Z 339.044,A -85,B 0,C 180,E1 -14253.846,E2 -14253.846} C_VEL
LIN {X 0,Y 340.703,Z 339.048,A -85,B 0,C 180,E1 -14256.741,E2 -14256.741} C_VEL
LIN {X 0,Y 340.686,Z 339.046,A -85,B 0,C 180,E1 -14260.246,E2 -14260.246} C_VEL
LIN {X 0,Y 340.666,Z 339.047,A -85,B 0,C 180,E1 -14263.775,E2 -14263.775} C_VEL
LIN {X 0,Y 340.674,Z 339.049,A -85,B 0,C 180,E1 -14267.095,E2 -14267.095} C_VEL
LIN {X 0,Y 340.697,Z 339.045,A -85,B 0,C 180,E1 -14270.247,E2 -14270.247} C_VEL
LIN {X 0,Y 340.709,Z 339.042,A -85,B 0,C 180,E1 -14273.558,E2 -14273.558} C_VEL
LIN {X 0,Y 340.69,Z 339.046,A -85,B 0,C 180,E1 -14276.153,E2 -14276.153} C_VEL
LIN {X 0,Y 340.738,Z 339.041,A -85,B 0,C 180,E1 -14280.329,E2 -14280.329} C_VEL
LIN {X 0,Y 340.8,Z 339.033,A -85,B 0,C 180,E1 -14283.02,E2 -14283.02} C_VEL
LIN {X 0,Y 340.727,Z 339.042,A -85,B 0,C 180,E1 -14286.927,E2 -14286.927} C_VEL
LIN {X 0,Y 340.788,Z 339.036,A -85,B 0,C 180,E1 -14290.733,E2 -14290.733} C_VEL
LIN {X 0,Y 340.783,Z 339.033,A -85,B 0,C 180,E1 -14293.219,E2 -14293.219} C_VEL
LIN {X 0,Y 340.841,Z 339.028,A -85,B 0,C 180,E1 -14296.89,E2 -14296.89} C_VEL
LIN {X 0,Y 340.926,Z 339.02,A -85,B 0,C 180,E1 -14300.508,E2 -14300.508} C_VEL
LIN {X 0,Y 341.073,Z 338.998,A -85,B 0,C 180,E1 -14302.898,E2 -14302.898} C_VEL
LIN {X 0,Y 341.167,Z 338.985,A -85,B 0,C 180,E1 -14307.639,E2 -14307.639} C_VEL
LIN {X 0,Y 341.294,Z 338.971,A -85,B 0,C 180,E1 -14310,E2 -14310} C_VEL
LIN {X 0,Y 341.167,Z 338.99,A -85,B 0,C 180,E1 -14312.361,E2 -14312.361} C_VEL
LIN {X 0,Y 341.073,Z 338.997,A -85,B 0,C 180,E1 -14317.102,E2 -14317.102} C_VEL
LIN {X 0,Y 340.869,Z 339.024,A -85,B 0,C 180,E1 -14320.694,E2 -14320.694} C_VEL
LIN {X 0,Y 340.86,Z 339.028,A -85,B 0,C 180,E1 -14324.325,E2 -14324.325} C_VEL
LIN {X 0,Y 340.836,Z 339.03,A -85,B 0,C 180,E1 -14328.467,E2 -14328.467} C_VEL
LIN {X 0,Y 340.752,Z 339.039,A -85,B 0,C 180,E1 -14331.857,E2 -14331.857} C_VEL
LIN {X 0,Y 340.771,Z 339.036,A -85,B 0,C 180,E1 -14335.665,E2 -14335.665} C_VEL
LIN {X 0,Y 340.727,Z 339.044,A -85,B 0,C 180,E1 -14338.321,E2 -14338.321} C_VEL
LIN {X 0,Y 340.696,Z 339.043,A -85,B 0,C 180,E1 -14341.045,E2 -14341.045} C_VEL
LIN {X 0,Y 340.717,Z 339.041,A -85,B 0,C 180,E1 -14345.279,E2 -14345.279} C_VEL
LIN {X 0,Y 340.71,Z 339.045,A -85,B 0,C 180,E1 -14348.387,E2 -14348.387} C_VEL
LIN {X 0,Y 340.698,Z 339.049,A -85,B 0,C 180,E1 -14352.046,E2 -14352.046} C_VEL
LIN {X 0,Y 340.652,Z 339.053,A -85,B 0,C 180,E1 -14356.228,E2 -14356.228} C_VEL
LIN {X 0,Y 340.688,Z 339.048,A -85,B 0,C 180,E1 -14359.754,E2 -14359.754} C_VEL
LIN {X 0,Y 340.69,Z 339.043,A -85,B 0,C 180,E1 -14362.841,E2 -14362.841} C_VEL
LIN {X 0,Y 340.035,Z 339.13,A -85,B 0,C 180,E1 -14363.827,E2 -14363.827} C_VEL
LIN {X 0,Y 337.17,Z 339.484,A -85,B 0,C 180,E1 -14365.43,E2 -14365.43} C_VEL
LIN {X 0,Y 334.741,Z 339.785,A -85,B 0,C 180,E1 -14366.729,E2 -14366.729} C_VEL
LIN {X 0,Y 333.709,Z 339.918,A -85,B 0,C 180,E1 -14367.734,E2 -14367.734} C_VEL
LIN {X 0,Y 333.631,Z 339.926,A -85,B 0,C 180,E1 -14368.075,E2 -14368.075} C_VEL
LIN {X 0,Y 333.766,Z 339.908,A -85,B 0,C 180,E1 -14370.543,E2 -14370.543} C_VEL
LIN {X 0,Y 340.327,Z 360.566,A -85,B 0,C 180,E1 -14371.45,E2 -14371.45} C_VEL
LIN {X 0,Y 338.673,Z 427.181,A -85,B 0,C 180,E1 -14373.29,E2 -14373.29} C_VEL
LIN {X 0,Y 338.434,Z 439.828,A -85,B 0,C 180,E1 -14373.865,E2 -14373.865} C_VEL
LIN {X 0,Y 337.871,Z 453.784,A -85,B 0,C 180,E1 -14374.76,E2 -14374.76} C_VEL
LIN {X 0,Y 337.361,Z 464.929,A -85,B 0,C 180,E1 -14375.705,E2 -14375.705} C_VEL
LIN {X 0,Y 336.653,Z 476.645,A -85,B 0,C 180,E1 -14376.957,E2 -14376.957} C_VEL
LIN {X 0,Y 335.93,Z 487.263,A -85,B 0,C 180,E1 -14378.363,E2 -14378.363} C_VEL
LIN {X 0,Y 335.138,Z 497.659,A -85,B 0,C 180,E1 -14380.077,E2 -14380.077} C_VEL
LIN {X 0,Y 334.478,Z 506.732,A -85,B 0,C 180,E1 -14381.946,E2 -14381.946} C_VEL
LIN {X 0,Y 333.968,Z 513.961,A -85,B 0,C 180,E1 -14383.81,E2 -14383.81} C_VEL
LIN {X 0,Y 333.633,Z 519.777,A -85,B 0,C 180,E1 -14385.697,E2 -14385.697} C_VEL
LIN {X 0,Y 333.369,Z 524.726,A -85,B 0,C 180,E1 -14387.83,E2 -14387.83} C_VEL
LIN {X 0,Y 333.308,Z 526.936,A -85,B 0,C 180,E1 -14389.061,E2 -14389.061} C_VEL
LIN {X 0,Y 333.333,Z 528.622,A -85,B 0,C 180,E1 -14390.29,E2 -14390.29} C_VEL
LIN {X 0,Y 333.504,Z 530.294,A -85,B 0,C 180,E1 -14392.076,E2 -14392.076} C_VEL
LIN {X 0,Y 333.689,Z 531.052,A -85,B 0,C 180,E1 -14393.956,E2 -14393.956} C_VEL
LIN {X 0,Y 333.779,Z 531.002,A -85,B 0,C 180,E1 -14395.169,E2 -14395.169} C_VEL
LIN {X 0,Y 334.137,Z 530.519,A -85,B 0,C 180,E1 -14396.383,E2 -14396.383} C_VEL
LIN {X 0,Y 334.476,Z 529.578,A -85,B 0,C 180,E1 -14397.592,E2 -14397.592} C_VEL
LIN {X 0,Y 334.93,Z 528.204,A -85,B 0,C 180,E1 -14398.798,E2 -14398.798} C_VEL
LIN {X 0,Y 335.705,Z 525.31,A -85,B 0,C 180,E1 -14400.6,E2 -14400.6} C_VEL
LIN {X 0,Y 336.68,Z 521.315,A -85,B 0,C 180,E1 -14402.393,E2 -14402.393} C_VEL
LIN {X 0,Y 337.829,Z 516.116,A -85,B 0,C 180,E1 -14404.176,E2 -14404.176} C_VEL
LIN {X 0,Y 339.255,Z 508.985,A -85,B 0,C 180,E1 -14406.08,E2 -14406.08} C_VEL
LIN {X 0,Y 340.687,Z 501.36,A -85,B 0,C 180,E1 -14407.706,E2 -14407.706} C_VEL
LIN {X 0,Y 342.029,Z 493.003,A -85,B 0,C 180,E1 -14409.164,E2 -14409.164} C_VEL
LIN {X 0,Y 343.546,Z 482.625,A -85,B 0,C 180,E1 -14410.61,E2 -14410.61} C_VEL
LIN {X 0,Y 344.769,Z 472.45,A -85,B 0,C 180,E1 -14411.763,E2 -14411.763} C_VEL
LIN {X 0,Y 345.972,Z 461.366,A -85,B 0,C 180,E1 -14412.763,E2 -14412.763} C_VEL
LIN {X 0,Y 346.906,Z 448.15,A -85,B 0,C 180,E1 -14413.697,E2 -14413.697} C_VEL
LIN {X 0,Y 347.513,Z 435.228,A -85,B 0,C 180,E1 -14414.344,E2 -14414.344} C_VEL
LIN {X 0,Y 348.578,Z 408.451,A -85,B 0,C 180,E1 -14415.232,E2 -14415.232} C_VEL
LIN {X 0,Y 350.849,Z 370.113,A -85,B 0,C 180,E1 -14416.436,E2 -14416.436} C_VEL
LIN {X 0,Y 345.119,Z 359.068,A -85,B 0,C 180,E1 -14417.681,E2 -14417.681} C_VEL
LIN {X 0,Y 338.937,Z 348.794,A -85,B 0,C 180,E1 -14419.108,E2 -14419.108} C_VEL
LIN {X 0,Y 336.746,Z 345.372,A -85,B 0,C 180,E1 -14419.653,E2 -14419.653} C_VEL
LIN {X 0,Y 336.146,Z 344.47,A -85,B 0,C 180,E1 -14419.805,E2 -14419.805} C_VEL
LIN {X 0,Y 334.438,Z 342.349,A -85,B 0,C 180,E1 -14420.221,E2 -14420.221} C_VEL
LIN {X 0,Y 333.675,Z 339.922,A -85,B 0,C 180,E1 -14420.505,E2 -14420.505} C_VEL
LIN {X 0,Y 333.645,Z 339.924,A -85,B 0,C 180,E1 -14423.593,E2 -14423.593} C_VEL
LIN {X 0,Y 333.633,Z 339.928,A -85,B 0,C 180,E1 -14426.256,E2 -14426.256} C_VEL
LIN {X 0,Y 333.635,Z 339.925,A -85,B 0,C 180,E1 -14428.98,E2 -14428.98} C_VEL
LIN {X 0,Y 333.648,Z 339.925,A -85,B 0,C 180,E1 -14432.587,E2 -14432.587} C_VEL
LIN {X 0,Y 333.677,Z 339.917,A -85,B 0,C 180,E1 -14436.139,E2 -14436.139} C_VEL
LIN {X 0,Y 333.623,Z 339.923,A -85,B 0,C 180,E1 -14439.196,E2 -14439.196} C_VEL
LIN {X 0,Y 333.631,Z 339.922,A -85,B 0,C 180,E1 -14442.499,E2 -14442.499} C_VEL
LIN {X 0,Y 333.598,Z 339.93,A -85,B 0,C 180,E1 -14445.955,E2 -14445.955} C_VEL
LIN {X 0,Y 333.606,Z 339.931,A -85,B 0,C 180,E1 -14449.324,E2 -14449.324} C_VEL
LIN {X 0,Y 333.666,Z 339.922,A -85,B 0,C 180,E1 -14453.168,E2 -14453.168} C_VEL
LIN {X 0,Y 333.751,Z 340.001,A -85,B 0,C 180,E1 -14455.556,E2 -14455.556} C_VEL
LIN {X 0,Y 337.759,Z 358.757,A -85,B 0,C 180,E1 -14459.696,E2 -14459.696} C_VEL
LIN {X 0,Y 338.906,Z 364.697,A -85,B 0,C 180,E1 -14460.963,E2 -14460.963} C_VEL
LIN {X 0,Y 338.77,Z 366.988,A -85,B 0,C 180,E1 -14461.363,E2 -14461.363} C_VEL
LIN {X 0,Y 339.735,Z 377.105,A -85,B 0,C 180,E1 -14462.237,E2 -14462.237} C_VEL
LIN {X 0,Y 341.602,Z 388.395,A -85,B 0,C 180,E1 -14462.998,E2 -14462.998} C_VEL
LIN {X 0,Y 344.151,Z 408.836,A -85,B 0,C 180,E1 -14464.208,E2 -14464.208} C_VEL
LIN {X 0,Y 346.089,Z 427.92,A -85,B 0,C 180,E1 -14465.209,E2 -14465.209} C_VEL
LIN {X 0,Y 347.274,Z 449.789,A -85,B 0,C 180,E1 -14466.181,E2 -14466.181} C_VEL
LIN {X 0,Y 344.516,Z 502.715,A -85,B 0,C 180,E1 -14467.827,E2 -14467.827} C_VEL
LIN {X 0,Y 343.28,Z 516.374,A -85,B 0,C 180,E1 -14468.454,E2 -14468.454} C_VEL
LIN {X 0,Y 341.802,Z 528.619,A -85,B 0,C 180,E1 -14469.225,E2 -14469.225} C_VEL
LIN {X 0,Y 340.065,Z 540.786,A -85,B 0,C 180,E1 -14470.219,E2 -14470.219} C_VEL
LIN {X 0,Y 338.448,Z 551.959,A -85,B 0,C 180,E1 -14471.381,E2 -14471.381} C_VEL
LIN {X 0,Y 336.636,Z 563.245,A -85,B 0,C 180,E1 -14472.849,E2 -14472.849} C_VEL
LIN {X 0,Y 335.159,Z 573.268,A -85,B 0,C 180,E1 -14474.453,E2 -14474.453} C_VEL
LIN {X 0,Y 333.954,Z 582.51,A -85,B 0,C 180,E1 -14476.305,E2 -14476.305} C_VEL
LIN {X 0,Y 333.162,Z 589.896,A -85,B 0,C 180,E1 -14478.131,E2 -14478.131} C_VEL
LIN {X 0,Y 332.616,Z 596.76,A -85,B 0,C 180,E1 -14480.268,E2 -14480.268} C_VEL
LIN {X 0,Y 332.495,Z 601.315,A -85,B 0,C 180,E1 -14482.103,E2 -14482.103} C_VEL
LIN {X 0,Y 332.632,Z 604.763,A -85,B 0,C 180,E1 -14483.936,E2 -14483.936} C_VEL
LIN {X 0,Y 332.755,Z 606.466,A -85,B 0,C 180,E1 -14485.153,E2 -14485.153} C_VEL
LIN {X 0,Y 332.932,Z 607.74,A -85,B 0,C 180,E1 -14486.369,E2 -14486.369} C_VEL
LIN {X 0,Y 333.116,Z 610.067,A -85,B 0,C 180,E1 -14490,E2 -14490} C_VEL
LIN {X 0,Y 332.983,Z 610.242,A -85,B 0,C 180,E1 -14491.209,E2 -14491.209} C_VEL
LIN {X 0,Y 332.903,Z 609.971,A -85,B 0,C 180,E1 -14492.42,E2 -14492.42} C_VEL
LIN {X 0,Y 332.838,Z 609.261,A -85,B 0,C 180,E1 -14493.632,E2 -14493.632} C_VEL
LIN {X 0,Y 332.635,Z 608.079,A -85,B 0,C 180,E1 -14494.848,E2 -14494.848} C_VEL
LIN {X 0,Y 332.498,Z 605.64,A -85,B 0,C 180,E1 -14496.563,E2 -14496.563} C_VEL
LIN {X 0,Y 332.452,Z 601.771,A -85,B 0,C 180,E1 -14498.51,E2 -14498.51} C_VEL
LIN {X 0,Y 332.644,Z 596.982,A -85,B 0,C 180,E1 -14500.345,E2 -14500.345} C_VEL
LIN {X 0,Y 333.366,Z 589.84,A -85,B 0,C 180,E1 -14502.479,E2 -14502.479} C_VEL
LIN {X 0,Y 334.406,Z 582.233,A -85,B 0,C 180,E1 -14504.297,E2 -14504.297} C_VEL
LIN {X 0,Y 335.444,Z 574.631,A -85,B 0,C 180,E1 -14505.805,E2 -14505.805} C_VEL
LIN {X 0,Y 337.046,Z 564.634,A -85,B 0,C 180,E1 -14507.442,E2 -14507.442} C_VEL
LIN {X 0,Y 338.974,Z 553.559,A -85,B 0,C 180,E1 -14508.902,E2 -14508.902} C_VEL
LIN {X 0,Y 340.961,Z 541.385,A -85,B 0,C 180,E1 -14510.197,E2 -14510.197} C_VEL
LIN {X 0,Y 343.029,Z 527.727,A -85,B 0,C 180,E1 -14511.325,E2 -14511.325} C_VEL
LIN {X 0,Y 344.735,Z 514.496,A -85,B 0,C 180,E1 -14512.157,E2 -14512.157} C_VEL
LIN {X 0,Y 346.171,Z 499.442,A -85,B 0,C 180,E1 -14512.847,E2 -14512.847} C_VEL
LIN {X 0,Y 349.242,Z 449.005,A -85,B 0,C 180,E1 -14514.482,E2 -14514.482} C_VEL
LIN {X 0,Y 348.584,Z 432.512,A -85,B 0,C 180,E1 -14515.254,E2 -14515.254} C_VEL
LIN {X 0,Y 347.39,Z 418.846,A -85,B 0,C 180,E1 -14516.009,E2 -14516.009} C_VEL
LIN {X 0,Y 344.673,Z 400.241,A -85,B 0,C 180,E1 -14517.261,E2 -14517.261} C_VEL
LIN {X 0,Y 342.009,Z 386.785,A -85,B 0,C 180,E1 -14518.353,E2 -14518.353} C_VEL
LIN {X 0,Y 341.359,Z 382.998,A -85,B 0,C 180,E1 -14518.683,E2 -14518.683} C_VEL
LIN {X 0,Y 342.956,Z 374.846,A -85,B 0,C 180,E1 -14520.606,E2 -14520.606} C_VEL
LIN {X 0,Y 341.908,Z 368.344,A -85,B 0,C 180,E1 -14522.566,E2 -14522.566} C_VEL
LIN {X 0,Y 340.086,Z 360.306,A -85,B 0,C 180,E1 -14525.354,E2 -14525.354} C_VEL
LIN {X 0,Y 338.293,Z 354.216,A -85,B 0,C 180,E1 -14527.865,E2 -14527.865} C_VEL
LIN {X 0,Y 336.739,Z 349.267,A -85,B 0,C 180,E1 -14530.315,E2 -14530.315} C_VEL
LIN {X 0,Y 335.377,Z 345.099,A -85,B 0,C 180,E1 -14532.824,E2 -14532.824} C_VEL
LIN {X 0,Y 334.642,Z 342.921,A -85,B 0,C 180,E1 -14534.434,E2 -14534.434} C_VEL
LIN {X 0,Y 333.631,Z 339.928,A -85,B 0,C 180,E1 -14537.5,E2 -14537.5} C_VEL
LIN {X 0,Y 333.636,Z 339.926,A -85,B 0,C 180,E1 -14541.206,E2 -14541.206} C_VEL
LIN {X 0,Y 333.675,Z 339.921,A -85,B 0,C 180,E1 -14543.86,E2 -14543.86} C_VEL
LIN {X 0,Y 333.646,Z 339.926,A -85,B 0,C 180,E1 -14547.413,E2 -14547.413} C_VEL
LIN {X 0,Y 333.653,Z 339.958,A -85,B 0,C 180,E1 -14551.022,E2 -14551.022} C_VEL
LIN {X 0,Y 333.833,Z 340.901,A -85,B 0,C 180,E1 -14551.943,E2 -14551.943} C_VEL
LIN {X 0,Y 335.135,Z 343.475,A -85,B 0,C 180,E1 -14552.419,E2 -14552.419} C_VEL
LIN {X 0,Y 337.013,Z 345.263,A -85,B 0,C 180,E1 -14552.962,E2 -14552.962} C_VEL
LIN {X 0,Y 338.87,Z 348.564,A -85,B 0,C 180,E1 -14553.563,E2 -14553.563} C_VEL
LIN {X 0,Y 340.227,Z 350.244,A -85,B 0,C 180,E1 -14553.935,E2 -14553.935} C_VEL
LIN {X 0,Y 345.141,Z 357.95,A -85,B 0,C 180,E1 -14555.287,E2 -14555.287} C_VEL
LIN {X 0,Y 351.09,Z 368.775,A -85,B 0,C 180,E1 -14556.8,E2 -14556.8} C_VEL
LIN {X 0,Y 352.921,Z 372.573,A -85,B 0,C 180,E1 -14557.247,E2 -14557.247} C_VEL
LIN {X 0,Y 349.177,Z 424.66,A -85,B 0,C 180,E1 -14558.99,E2 -14558.99} C_VEL
LIN {X 0,Y 348.562,Z 440.905,A -85,B 0,C 180,E1 -14559.646,E2 -14559.646} C_VEL
LIN {X 0,Y 347.699,Z 454.375,A -85,B 0,C 180,E1 -14560.441,E2 -14560.441} C_VEL
LIN {X 0,Y 346.591,Z 466.403,A -85,B 0,C 180,E1 -14561.375,E2 -14561.375} C_VEL
LIN {X 0,Y 345.215,Z 477.872,A -85,B 0,C 180,E1 -14562.525,E2 -14562.525} C_VEL
LIN {X 0,Y 343.763,Z 488.302,A -85,B 0,C 180,E1 -14563.826,E2 -14563.826} C_VEL
LIN {X 0,Y 342.053,Z 498.361,A -85,B 0,C 180,E1 -14565.391,E2 -14565.391} C_VEL
LIN {X 0,Y 340.352,Z 507.498,A -85,B 0,C 180,E1 -14567.174,E2 -14567.174} C_VEL
LIN {X 0,Y 338.826,Z 514.622,A -85,B 0,C 180,E1 -14568.938,E2 -14568.938} C_VEL
LIN {X 0,Y 337.342,Z 521.134,A -85,B 0,C 180,E1 -14571.01,E2 -14571.01} C_VEL
LIN {X 0,Y 336.219,Z 525.377,A -85,B 0,C 180,E1 -14572.795,E2 -14572.795} C_VEL
LIN {X 0,Y 335.621,Z 527.553,A -85,B 0,C 180,E1 -14573.989,E2 -14573.989} C_VEL
LIN {X 0,Y 335.077,Z 529.279,A -85,B 0,C 180,E1 -14575.187,E2 -14575.187} C_VEL
LIN {X 0,Y 334.623,Z 530.575,A -85,B 0,C 180,E1 -14576.387,E2 -14576.387} C_VEL
LIN {X 0,Y 334.308,Z 531.394,A -85,B 0,C 180,E1 -14577.59,E2 -14577.59} C_VEL
LIN {X 0,Y 333.971,Z 531.803,A -85,B 0,C 180,E1 -14578.794,E2 -14578.794} C_VEL
LIN {X 0,Y 333.831,Z 531.783,A -85,B 0,C 180,E1 -14579.999,E2 -14579.999} C_VEL
LIN {X 0,Y 333.555,Z 531.354,A -85,B 0,C 180,E1 -14581.207,E2 -14581.207} C_VEL
LIN {X 0,Y 333.159,Z 530.487,A -85,B 0,C 180,E1 -14582.417,E2 -14582.417} C_VEL
LIN {X 0,Y 333.238,Z 529.164,A -85,B 0,C 180,E1 -14583.627,E2 -14583.627} C_VEL
LIN {X 0,Y 333.46,Z 526.34,A -85,B 0,C 180,E1 -14585.442,E2 -14585.442} C_VEL
LIN {X 0,Y 333.533,Z 522.475,A -85,B 0,C 180,E1 -14587.263,E2 -14587.263} C_VEL
LIN {X 0,Y 333.791,Z 517.439,A -85,B 0,C 180,E1 -14589.085,E2 -14589.085} C_VEL
LIN {X 0,Y 334.15,Z 511.047,A -85,B 0,C 180,E1 -14590.911,E2 -14590.911} C_VEL
LIN {X 0,Y 334.643,Z 503.071,A -85,B 0,C 180,E1 -14592.739,E2 -14592.739} C_VEL
LIN {X 0,Y 335.237,Z 494.968,A -85,B 0,C 180,E1 -14594.26,E2 -14594.26} C_VEL
LIN {X 0,Y 335.802,Z 485.116,A -85,B 0,C 180,E1 -14595.787,E2 -14595.787} C_VEL
LIN {X 0,Y 336.627,Z 472.858,A -85,B 0,C 180,E1 -14597.307,E2 -14597.307} C_VEL
LIN {X 0,Y 337.18,Z 462.134,A -85,B 0,C 180,E1 -14598.376,E2 -14598.376} C_VEL
LIN {X 0,Y 337.815,Z 449.502,A -85,B 0,C 180,E1 -14599.363,E2 -14599.363} C_VEL
LIN {X 0,Y 338.257,Z 435.827,A -85,B 0,C 180,E1 -14600.167,E2 -14600.167} C_VEL
LIN {X 0,Y 338.45,Z 421.975,A -85,B 0,C 180,E1 -14600.718,E2 -14600.718} C_VEL
LIN {X 0,Y 339.96,Z 359.517,A -85,B 0,C 180,E1 -14602.493,E2 -14602.493} C_VEL
LIN {X 0,Y 333.72,Z 339.914,A -85,B 0,C 180,E1 -14603.363,E2 -14603.363} C_VEL
LIN {X 0,Y 333.736,Z 339.911,A -85,B 0,C 180,E1 -14606.246,E2 -14606.246} C_VEL
LIN {X 0,Y 333.711,Z 339.918,A -85,B 0,C 180,E1 -14608.971,E2 -14608.971} C_VEL
LIN {X 0,Y 333.642,Z 339.925,A -85,B 0,C 180,E1 -14612.586,E2 -14612.586} C_VEL
LIN {X 0,Y 333.675,Z 339.919,A -85,B 0,C 180,E1 -14616.138,E2 -14616.138} C_VEL
LIN {X 0,Y 333.645,Z 339.924,A -85,B 0,C 180,E1 -14619.192,E2 -14619.192} C_VEL
LIN {X 0,Y 333.632,Z 339.927,A -85,B 0,C 180,E1 -14622.5,E2 -14622.5} C_VEL
LIN {X 0,Y 333.617,Z 339.925,A -85,B 0,C 180,E1 -14625.958,E2 -14625.958} C_VEL
LIN {X 0,Y 333.645,Z 339.923,A -85,B 0,C 180,E1 -14629.315,E2 -14629.315} C_VEL
LIN {X 0,Y 333.665,Z 339.921,A -85,B 0,C 180,E1 -14633.167,E2 -14633.167} C_VEL
LIN {X 0,Y 333.634,Z 339.928,A -85,B 0,C 180,E1 -14636.791,E2 -14636.791} C_VEL
LIN {X 0,Y 333.692,Z 339.916,A -85,B 0,C 180,E1 -14639.712,E2 -14639.712} C_VEL
LIN {X 0,Y 333.737,Z 339.914,A -85,B 0,C 180,E1 -14642.401,E2 -14642.401} C_VEL
LIN {X 0,Y 333.724,Z 339.913,A -85,B 0,C 180,E1 -14645.091,E2 -14645.091} C_VEL
LIN {X 0,Y 333.682,Z 339.919,A -85,B 0,C 180,E1 -14649.019,E2 -14649.019} C_VEL
LIN {X 0,Y 333.79,Z 339.903,A -85,B 0,C 180,E1 -14651.589,E2 -14651.589} C_VEL
LIN {X 0,Y 333.805,Z 339.902,A -85,B 0,C 180,E1 -14655.577,E2 -14655.577} C_VEL
LIN {X 0,Y 333.832,Z 339.899,A -85,B 0,C 180,E1 -14659.078,E2 -14659.078} C_VEL
LIN {X 0,Y 334.023,Z 339.878,A -85,B 0,C 180,E1 -14662.748,E2 -14662.748} C_VEL
LIN {X 0,Y 333.808,Z 339.902,A -85,B 0,C 180,E1 -14665.169,E2 -14665.169} C_VEL
LIN {X 0,Y 334.105,Z 339.865,A -85,B 0,C 180,E1 -14667.589,E2 -14667.589} C_VEL
LIN {X 0,Y 334.245,Z 339.849,A -85,B 0,C 180,E1 -14670,E2 -14670} C_VEL
LIN {X 0,Y 334.105,Z 339.87,A -85,B 0,C 180,E1 -14672.411,E2 -14672.411} C_VEL
LIN {X 0,Y 334.023,Z 339.875,A -85,B 0,C 180,E1 -14677.253,E2 -14677.253} C_VEL
LIN {X 0,Y 333.831,Z 339.899,A -85,B 0,C 180,E1 -14680.922,E2 -14680.922} C_VEL
LIN {X 0,Y 333.806,Z 339.904,A -85,B 0,C 180,E1 -14684.635,E2 -14684.635} C_VEL
LIN {X 0,Y 333.795,Z 339.905,A -85,B 0,C 180,E1 -14688.656,E2 -14688.656} C_VEL
LIN {X 0,Y 333.69,Z 339.921,A -85,B 0,C 180,E1 -14692.279,E2 -14692.279} C_VEL
LIN {X 0,Y 333.733,Z 339.916,A -85,B 0,C 180,E1 -14696.247,E2 -14696.247} C_VEL
LIN {X 0,Y 333.688,Z 339.916,A -85,B 0,C 180,E1 -14698.975,E2 -14698.975} C_VEL
LIN {X 0,Y 333.644,Z 339.924,A -85,B 0,C 180,E1 -14702.588,E2 -14702.588} C_VEL
LIN {X 0,Y 333.676,Z 339.923,A -85,B 0,C 180,E1 -14706.14,E2 -14706.14} C_VEL
LIN {X 0,Y 333.646,Z 339.922,A -85,B 0,C 180,E1 -14709.193,E2 -14709.193} C_VEL
LIN {X 0,Y 333.632,Z 339.925,A -85,B 0,C 180,E1 -14712.501,E2 -14712.501} C_VEL
LIN {X 0,Y 333.596,Z 339.933,A -85,B 0,C 180,E1 -14715.956,E2 -14715.956} C_VEL
LIN {X 0,Y 333.647,Z 339.922,A -85,B 0,C 180,E1 -14719.316,E2 -14719.316} C_VEL
LIN {X 0,Y 333.665,Z 339.919,A -85,B 0,C 180,E1 -14723.169,E2 -14723.169} C_VEL
LIN {X 0,Y 333.675,Z 339.919,A -85,B 0,C 180,E1 -14725.342,E2 -14725.342} C_VEL
LIN {X 0,Y 333.631,Z 339.926,A -85,B 0,C 180,E1 -14728.075,E2 -14728.075} C_VEL
LIN {X 0,Y 333.632,Z 340.654,A -85,B 0,C 180,E1 -14728.705,E2 -14728.705} C_VEL
LIN {X 0,Y 333.624,Z 342.464,A -85,B 0,C 180,E1 -14729.276,E2 -14729.276} C_VEL
LIN {X 0,Y 333.609,Z 345.026,A -85,B 0,C 180,E1 -14729.779,E2 -14729.779} C_VEL
LIN {X 0,Y 333.567,Z 349.843,A -85,B 0,C 180,E1 -14730.39,E2 -14730.39} C_VEL
LIN {X 0,Y 333.471,Z 357.487,A -85,B 0,C 180,E1 -14730.984,E2 -14730.984} C_VEL
LIN {X 0,Y 333.37,Z 363.605,A -85,B 0,C 180,E1 -14731.243,E2 -14731.243} C_VEL
LIN {X 0,Y 331.722,Z 427.29,A -85,B 0,C 180,E1 -14733.059,E2 -14733.059} C_VEL
LIN {X 0,Y 331.458,Z 440.13,A -85,B 0,C 180,E1 -14733.645,E2 -14733.645} C_VEL
LIN {X 0,Y 330.922,Z 453.739,A -85,B 0,C 180,E1 -14734.529,E2 -14734.529} C_VEL
LIN {X 0,Y 330.377,Z 465.098,A -85,B 0,C 180,E1 -14735.493,E2 -14735.493} C_VEL
LIN {X 0,Y 329.599,Z 477.659,A -85,B 0,C 180,E1 -14736.856,E2 -14736.856} C_VEL
LIN {X 0,Y 328.905,Z 487.7,A -85,B 0,C 180,E1 -14738.207,E2 -14738.207} C_VEL
LIN {X 0,Y 328.116,Z 498.196,A -85,B 0,C 180,E1 -14739.959,E2 -14739.959} C_VEL
LIN {X 0,Y 327.53,Z 505.993,A -85,B 0,C 180,E1 -14741.549,E2 -14741.549} C_VEL
LIN {X 0,Y 327,Z 513.557,A -85,B 0,C 180,E1 -14743.455,E2 -14743.455} C_VEL
LIN {X 0,Y 326.595,Z 520.125,A -85,B 0,C 180,E1 -14745.55,E2 -14745.55} C_VEL
LIN {X 0,Y 326.346,Z 524.94,A -85,B 0,C 180,E1 -14747.564,E2 -14747.564} C_VEL
LIN {X 0,Y 326.265,Z 527.258,A -85,B 0,C 180,E1 -14748.822,E2 -14748.822} C_VEL
LIN {X 0,Y 326.288,Z 529.13,A -85,B 0,C 180,E1 -14750.078,E2 -14750.078} C_VEL
LIN {X 0,Y 326.445,Z 531.095,A -85,B 0,C 180,E1 -14752.029,E2 -14752.029} C_VEL
LIN {X 0,Y 326.643,Z 531.967,A -85,B 0,C 180,E1 -14753.825,E2 -14753.825} C_VEL
LIN {X 0,Y 326.74,Z 532.042,A -85,B 0,C 180,E1 -14755.065,E2 -14755.065} C_VEL
LIN {X 0,Y 327.086,Z 531.666,A -85,B 0,C 180,E1 -14756.305,E2 -14756.305} C_VEL
LIN {X 0,Y 327.458,Z 530.894,A -85,B 0,C 180,E1 -14757.54,E2 -14757.54} C_VEL
LIN {X 0,Y 327.925,Z 529.646,A -85,B 0,C 180,E1 -14758.773,E2 -14758.773} C_VEL
LIN {X 0,Y 328.729,Z 526.95,A -85,B 0,C 180,E1 -14760.613,E2 -14760.613} C_VEL
LIN {X 0,Y 329.739,Z 523.182,A -85,B 0,C 180,E1 -14762.444,E2 -14762.444} C_VEL
LIN {X 0,Y 330.965,Z 518.25,A -85,B 0,C 180,E1 -14764.263,E2 -14764.263} C_VEL
LIN {X 0,Y 332.334,Z 512.017,A -85,B 0,C 180,E1 -14766.07,E2 -14766.07} C_VEL
LIN {X 0,Y 333.945,Z 504.164,A -85,B 0,C 180,E1 -14767.863,E2 -14767.863} C_VEL
LIN {X 0,Y 335.676,Z 494.368,A -85,B 0,C 180,E1 -14769.643,E2 -14769.643} C_VEL
LIN {X 0,Y 337.212,Z 484.78,A -85,B 0,C 180,E1 -14771.035,E2 -14771.035} C_VEL
LIN {X 0,Y 338.63,Z 474.188,A -85,B 0,C 180,E1 -14772.283,E2 -14772.283} C_VEL
LIN {X 0,Y 339.964,Z 462.507,A -85,B 0,C 180,E1 -14773.365,E2 -14773.365} C_VEL
LIN {X 0,Y 340.985,Z 449.173,A -85,B 0,C 180,E1 -14774.32,E2 -14774.32} C_VEL
LIN {X 0,Y 341.663,Z 435.542,A -85,B 0,C 180,E1 -14775.014,E2 -14775.014} C_VEL
LIN {X 0,Y 342.878,Z 408.653,A -85,B 0,C 180,E1 -14775.932,E2 -14775.932} C_VEL
LIN {X 0,Y 345.261,Z 372.83,A -85,B 0,C 180,E1 -14777.076,E2 -14777.076} C_VEL
LIN {X 0,Y 340.085,Z 362.844,A -85,B 0,C 180,E1 -14778.282,E2 -14778.282} C_VEL
LIN {X 0,Y 334.938,Z 354.143,A -85,B 0,C 180,E1 -14779.539,E2 -14779.539} C_VEL
LIN {X 0,Y 331.792,Z 349.487,A -85,B 0,C 180,E1 -14780.342,E2 -14780.342} C_VEL
LIN {X 0,Y 329.796,Z 346.195,A -85,B 0,C 180,E1 -14780.894,E2 -14780.894} C_VEL
LIN {X 0,Y 327.331,Z 343.137,A -85,B 0,C 180,E1 -14781.573,E2 -14781.573} C_VEL
LIN {X 0,Y 326.621,Z 340.807,A -85,B 0,C 180,E1 -14781.874,E2 -14781.874} C_VEL
LIN {X 0,Y 326.604,Z 340.805,A -85,B 0,C 180,E1 -14785.492,E2 -14785.492} C_VEL
LIN {X 0,Y 326.595,Z 340.806,A -85,B 0,C 180,E1 -14788.257,E2 -14788.257} C_VEL
LIN {X 0,Y 326.577,Z 340.806,A -85,B 0,C 180,E1 -14791.097,E2 -14791.097} C_VEL
LIN {X 0,Y 326.61,Z 340.8,A -85,B 0,C 180,E1 -14794.02,E2 -14794.02} C_VEL
LIN {X 0,Y 326.625,Z 340.795,A -85,B 0,C 180,E1 -14797.237,E2 -14797.237} C_VEL
LIN {X 0,Y 326.547,Z 340.803,A -85,B 0,C 180,E1 -14801.124,E2 -14801.124} C_VEL
LIN {X 0,Y 326.563,Z 340.806,A -85,B 0,C 180,E1 -14803.526,E2 -14803.526} C_VEL
LIN {X 0,Y 326.577,Z 340.805,A -85,B 0,C 180,E1 -14807.029,E2 -14807.029} C_VEL
LIN {X 0,Y 326.586,Z 340.805,A -85,B 0,C 180,E1 -14811.386,E2 -14811.386} C_VEL
LIN {X 0,Y 326.707,Z 340.898,A -85,B 0,C 180,E1 -14815.316,E2 -14815.316} C_VEL
LIN {X 0,Y 330.341,Z 357.888,A -85,B 0,C 180,E1 -14819.117,E2 -14819.117} C_VEL
LIN {X 0,Y 333.361,Z 369.015,A -85,B 0,C 180,E1 -14820.64,E2 -14820.64} C_VEL
LIN {X 0,Y 334.064,Z 376.135,A -85,B 0,C 180,E1 -14821.274,E2 -14821.274} C_VEL
LIN {X 0,Y 336.279,Z 391.067,A -85,B 0,C 180,E1 -14822.327,E2 -14822.327} C_VEL
LIN {X 0,Y 338.506,Z 409.453,A -85,B 0,C 180,E1 -14823.461,E2 -14823.461} C_VEL
LIN {X 0,Y 340.347,Z 429.154,A -85,B 0,C 180,E1 -14824.543,E2 -14824.543} C_VEL
LIN {X 0,Y 341.406,Z 450.515,A -85,B 0,C 180,E1 -14825.526,E2 -14825.526} C_VEL
LIN {X 0,Y 338.453,Z 502.645,A -85,B 0,C 180,E1 -14827.207,E2 -14827.207} C_VEL
LIN {X 0,Y 337.071,Z 516.472,A -85,B 0,C 180,E1 -14827.876,E2 -14827.876} C_VEL
LIN {X 0,Y 335.26,Z 530.213,A -85,B 0,C 180,E1 -14828.801,E2 -14828.801} C_VEL
LIN {X 0,Y 333.452,Z 541.739,A -85,B 0,C 180,E1 -14829.81,E2 -14829.81} C_VEL
LIN {X 0,Y 331.572,Z 553.704,A -85,B 0,C 180,E1 -14831.141,E2 -14831.141} C_VEL
LIN {X 0,Y 329.702,Z 564.538,A -85,B 0,C 180,E1 -14832.637,E2 -14832.637} C_VEL
LIN {X 0,Y 328.247,Z 573.552,A -85,B 0,C 180,E1 -14834.182,E2 -14834.182} C_VEL
LIN {X 0,Y 327.032,Z 582.286,A -85,B 0,C 180,E1 -14836.009,E2 -14836.009} C_VEL
LIN {X 0,Y 326.151,Z 589.551,A -85,B 0,C 180,E1 -14837.872,E2 -14837.872} C_VEL
LIN {X 0,Y 325.652,Z 594.495,A -85,B 0,C 180,E1 -14839.429,E2 -14839.429} C_VEL
LIN {X 0,Y 325.453,Z 599.329,A -85,B 0,C 180,E1 -14841.305,E2 -14841.305} C_VEL
LIN {X 0,Y 325.512,Z 603.267,A -85,B 0,C 180,E1 -14843.303,E2 -14843.303} C_VEL
LIN {X 0,Y 325.658,Z 605.7,A -85,B 0,C 180,E1 -14845.048,E2 -14845.048} C_VEL
LIN {X 0,Y 325.855,Z 606.913,A -85,B 0,C 180,E1 -14846.29,E2 -14846.29} C_VEL
LIN {X 0,Y 326.069,Z 608.251,A -85,B 0,C 180,E1 -14848.765,E2 -14848.765} C_VEL
LIN {X 0,Y 326.093,Z 609.008,A -85,B 0,C 180,E1 -14850,E2 -14850} C_VEL
LIN {X 0,Y 325.943,Z 609.276,A -85,B 0,C 180,E1 -14851.235,E2 -14851.235} C_VEL
LIN {X 0,Y 325.854,Z 609.053,A -85,B 0,C 180,E1 -14852.472,E2 -14852.472} C_VEL
LIN {X 0,Y 325.763,Z 608.386,A -85,B 0,C 180,E1 -14853.711,E2 -14853.711} C_VEL
LIN {X 0,Y 325.547,Z 607.268,A -85,B 0,C 180,E1 -14854.954,E2 -14854.954} C_VEL
LIN {X 0,Y 325.414,Z 605.156,A -85,B 0,C 180,E1 -14856.549,E2 -14856.549} C_VEL
LIN {X 0,Y 325.369,Z 601.149,A -85,B 0,C 180,E1 -14858.696,E2 -14858.696} C_VEL
LIN {X 0,Y 325.59,Z 596.486,A -85,B 0,C 180,E1 -14860.572,E2 -14860.572} C_VEL
LIN {X 0,Y 326.394,Z 589.545,A -85,B 0,C 180,E1 -14862.75,E2 -14862.75} C_VEL
LIN {X 0,Y 327.49,Z 582.112,A -85,B 0,C 180,E1 -14864.605,E2 -14864.605} C_VEL
LIN {X 0,Y 328.878,Z 573.074,A -85,B 0,C 180,E1 -14866.448,E2 -14866.448} C_VEL
LIN {X 0,Y 330.705,Z 562.994,A -85,B 0,C 180,E1 -14868.108,E2 -14868.108} C_VEL
LIN {X 0,Y 332.972,Z 550.652,A -85,B 0,C 180,E1 -14869.737,E2 -14869.737} C_VEL
LIN {X 0,Y 335.111,Z 538.064,A -85,B 0,C 180,E1 -14871.048,E2 -14871.048} C_VEL
LIN {X 0,Y 337.114,Z 525.915,A -85,B 0,C 180,E1 -14872.04,E2 -14872.04} C_VEL
LIN {X 0,Y 338.919,Z 512.582,A -85,B 0,C 180,E1 -14872.88,E2 -14872.88} C_VEL
LIN {X 0,Y 340.361,Z 498.436,A -85,B 0,C 180,E1 -14873.542,E2 -14873.542} C_VEL
LIN {X 0,Y 343.543,Z 449.178,A -85,B 0,C 180,E1 -14875.205,E2 -14875.205} C_VEL
LIN {X 0,Y 343.046,Z 433.932,A -85,B 0,C 180,E1 -14875.947,E2 -14875.947} C_VEL
LIN {X 0,Y 341.95,Z 420.36,A -85,B 0,C 180,E1 -14876.729,E2 -14876.729} C_VEL
LIN {X 0,Y 339.515,Z 402.767,A -85,B 0,C 180,E1 -14877.971,E2 -14877.971} C_VEL
LIN {X 0,Y 337.249,Z 390.28,A -85,B 0,C 180,E1 -14879.016,E2 -14879.016} C_VEL
LIN {X 0,Y 335.525,Z 381.158,A -85,B 0,C 180,E1 -14879.876,E2 -14879.876} C_VEL
LIN {X 0,Y 336.351,Z 377.594,A -85,B 0,C 180,E1 -14880.747,E2 -14880.747} C_VEL
LIN {X 0,Y 335.747,Z 372.685,A -85,B 0,C 180,E1 -14882.229,E2 -14882.229} C_VEL
LIN {X 0,Y 334.145,Z 364.996,A -85,B 0,C 180,E1 -14884.886,E2 -14884.886} C_VEL
LIN {X 0,Y 332.717,Z 359.636,A -85,B 0,C 180,E1 -14887.05,E2 -14887.05} C_VEL
LIN {X 0,Y 330.791,Z 353.33,A -85,B 0,C 180,E1 -14890.105,E2 -14890.105} C_VEL
LIN {X 0,Y 329.014,Z 348.048,A -85,B 0,C 180,E1 -14893.425,E2 -14893.425} C_VEL
LIN {X 0,Y 327.74,Z 344.357,A -85,B 0,C 180,E1 -14896.669,E2 -14896.669} C_VEL
LIN {X 0,Y 326.837,Z 342.153,A -85,B 0,C 180,E1 -14899.827,E2 -14899.827} C_VEL
LIN {X 0,Y 326.643,Z 341.052,A -85,B 0,C 180,E1 -14902.954,E2 -14902.954} C_VEL
LIN {X 0,Y 326.659,Z 340.963,A -85,B 0,C 180,E1 -14904.842,E2 -14904.842} C_VEL
LIN {X 0,Y 326.748,Z 341.619,A -85,B 0,C 180,E1 -14907.471,E2 -14907.471} C_VEL
LIN {X 0,Y 327.397,Z 343.214,A -85,B 0,C 180,E1 -14910.397,E2 -14910.397} C_VEL
LIN {X 0,Y 329.927,Z 346.292,A -85,B 0,C 180,E1 -14911.327,E2 -14911.327} C_VEL
LIN {X 0,Y 330.753,Z 347.515,A -85,B 0,C 180,E1 -14911.622,E2 -14911.622} C_VEL
LIN {X 0,Y 332.931,Z 350.499,A -85,B 0,C 180,E1 -14912.357,E2 -14912.357} C_VEL
LIN {X 0,Y 333.818,Z 351.753,A -85,B 0,C 180,E1 -14912.647,E2 -14912.647} C_VEL
LIN {X 0,Y 337.017,Z 356.719,A -85,B 0,C 180,E1 -14913.658,E2 -14913.658} C_VEL
LIN {X 0,Y 340.014,Z 361.417,A -85,B 0,C 180,E1 -14914.528,E2 -14914.528} C_VEL
LIN {X 0,Y 344.855,Z 369.967,A -85,B 0,C 180,E1 -14915.852,E2 -14915.852} C_VEL
LIN {X 0,Y 347.46,Z 375.188,A -85,B 0,C 180,E1 -14916.537,E2 -14916.537} C_VEL
LIN {X 0,Y 343.515,Z 426.862,A -85,B 0,C 180,E1 -14918.332,E2 -14918.332} C_VEL
LIN {X 0,Y 342.864,Z 442.199,A -85,B 0,C 180,E1 -14918.978,E2 -14918.978} C_VEL
LIN {X 0,Y 341.916,Z 455.496,A -85,B 0,C 180,E1 -14919.782,E2 -14919.782} C_VEL
LIN {X 0,Y 340.731,Z 467.432,A -85,B 0,C 180,E1 -14920.729,E2 -14920.729} C_VEL
LIN {X 0,Y 339.265,Z 478.864,A -85,B 0,C 180,E1 -14921.896,E2 -14921.896} C_VEL
LIN {X 0,Y 337.701,Z 489.16,A -85,B 0,C 180,E1 -14923.2,E2 -14923.2} C_VEL
LIN {X 0,Y 335.91,Z 499.153,A -85,B 0,C 180,E1 -14924.777,E2 -14924.777} C_VEL
LIN {X 0,Y 334.036,Z 508.45,A -85,B 0,C 180,E1 -14926.618,E2 -14926.618} C_VEL
LIN {X 0,Y 332.373,Z 515.593,A -85,B 0,C 180,E1 -14928.411,E2 -14928.411} C_VEL
LIN {X 0,Y 330.974,Z 521.268,A -85,B 0,C 180,E1 -14930.219,E2 -14930.219} C_VEL
LIN {X 0,Y 329.725,Z 525.705,A -85,B 0,C 180,E1 -14932.036,E2 -14932.036} C_VEL
LIN {X 0,Y 328.728,Z 529.01,A -85,B 0,C 180,E1 -14933.863,E2 -14933.863} C_VEL
LIN {X 0,Y 328.138,Z 530.651,A -85,B 0,C 180,E1 -14935.085,E2 -14935.085} C_VEL
LIN {X 0,Y 327.668,Z 531.813,A -85,B 0,C 180,E1 -14936.31,E2 -14936.31} C_VEL
LIN {X 0,Y 327.315,Z 532.535,A -85,B 0,C 180,E1 -14937.538,E2 -14937.538} C_VEL
LIN {X 0,Y 326.952,Z 532.861,A -85,B 0,C 180,E1 -14938.768,E2 -14938.768} C_VEL
LIN {X 0,Y 326.807,Z 532.737,A -85,B 0,C 180,E1 -14939.999,E2 -14939.999} C_VEL
LIN {X 0,Y 326.488,Z 532.184,A -85,B 0,C 180,E1 -14941.233,E2 -14941.233} C_VEL
LIN {X 0,Y 326.104,Z 531.232,A -85,B 0,C 180,E1 -14942.47,E2 -14942.47} C_VEL
LIN {X 0,Y 326.202,Z 529.817,A -85,B 0,C 180,E1 -14943.705,E2 -14943.705} C_VEL
LIN {X 0,Y 326.416,Z 526.834,A -85,B 0,C 180,E1 -14945.559,E2 -14945.559} C_VEL
LIN {X 0,Y 326.486,Z 522.79,A -85,B 0,C 180,E1 -14947.42,E2 -14947.42} C_VEL
LIN {X 0,Y 326.772,Z 516.519,A -85,B 0,C 180,E1 -14949.594,E2 -14949.594} C_VEL
LIN {X 0,Y 327.189,Z 509.682,A -85,B 0,C 180,E1 -14951.46,E2 -14951.46} C_VEL
LIN {X 0,Y 327.765,Z 501.13,A -85,B 0,C 180,E1 -14953.326,E2 -14953.326} C_VEL
LIN {X 0,Y 328.441,Z 491.093,A -85,B 0,C 180,E1 -14955.098,E2 -14955.098} C_VEL
LIN {X 0,Y 329.141,Z 480.565,A -85,B 0,C 180,E1 -14956.593,E2 -14956.593} C_VEL
LIN {X 0,Y 329.863,Z 468.348,A -85,B 0,C 180,E1 -14957.994,E2 -14957.994} C_VEL
LIN {X 0,Y 330.464,Z 456.189,A -85,B 0,C 180,E1 -14959.085,E2 -14959.085} C_VEL
LIN {X 0,Y 331.097,Z 442.666,A -85,B 0,C 180,E1 -14960.015,E2 -14960.015} C_VEL
LIN {X 0,Y 331.382,Z 428.922,A -85,B 0,C 180,E1 -14960.685,E2 -14960.685} C_VEL
LIN {X 0,Y 331.873,Z 401.006,A -85,B 0,C 180,E1 -14961.547,E2 -14961.547} C_VEL
LIN {X 0,Y 333.003,Z 360.868,A -85,B 0,C 180,E1 -14962.727,E2 -14962.727} C_VEL
LIN {X 0,Y 326.689,Z 340.788,A -85,B 0,C 180,E1 -14963.632,E2 -14963.632} C_VEL
LIN {X 0,Y 326.685,Z 340.794,A -85,B 0,C 180,E1 -14966.857,E2 -14966.857} C_VEL
LIN {X 0,Y 326.638,Z 340.798,A -85,B 0,C 180,E1 -14970.611,E2 -14970.611} C_VEL
LIN {X 0,Y 326.606,Z 340.799,A -85,B 0,C 180,E1 -14974.019,E2 -14974.019} C_VEL
LIN {X 0,Y 326.626,Z 340.798,A -85,B 0,C 180,E1 -14977.238,E2 -14977.238} C_VEL
LIN {X 0,Y 326.576,Z 340.805,A -85,B 0,C 180,E1 -14981.131,E2 -14981.131} C_VEL
LIN {X 0,Y 326.555,Z 340.811,A -85,B 0,C 180,E1 -14984.748,E2 -14984.748} C_VEL
LIN {X 0,Y 326.574,Z 340.803,A -85,B 0,C 180,E1 -14988.154,E2 -14988.154} C_VEL
LIN {X 0,Y 326.622,Z 340.797,A -85,B 0,C 180,E1 -14991.391,E2 -14991.391} C_VEL
LIN {X 0,Y 326.618,Z 340.801,A -85,B 0,C 180,E1 -14994.851,E2 -14994.851} C_VEL
LIN {X 0,Y 326.605,Z 340.799,A -85,B 0,C 180,E1 -14997.455,E2 -14997.455} C_VEL
LIN {X 0,Y 326.645,Z 340.797,A -85,B 0,C 180,E1 -15000.339,E2 -15000.339} C_VEL
LIN {X 0,Y 326.687,Z 340.793,A -85,B 0,C 180,E1 -15004.516,E2 -15004.516} C_VEL
LIN {X 0,Y 326.646,Z 340.799,A -85,B 0,C 180,E1 -15008.545,E2 -15008.545} C_VEL
LIN {X 0,Y 326.741,Z 340.782,A -85,B 0,C 180,E1 -15011.177,E2 -15011.177} C_VEL
LIN {X 0,Y 326.76,Z 340.779,A -85,B 0,C 180,E1 -15015.433,E2 -15015.433} C_VEL
LIN {X 0,Y 326.768,Z 340.781,A -85,B 0,C 180,E1 -15018.839,E2 -15018.839} C_VEL
LIN {X 0,Y 326.977,Z 340.757,A -85,B 0,C 180,E1 -15022.59,E2 -15022.59} C_VEL
LIN {X 0,Y 326.775,Z 340.778,A -85,B 0,C 180,E1 -15025.065,E2 -15025.065} C_VEL
LIN {X 0,Y 327.045,Z 340.744,A -85,B 0,C 180,E1 -15027.537,E2 -15027.537} C_VEL
LIN {X 0,Y 327.196,Z 340.727,A -85,B 0,C 180,E1 -15030,E2 -15030} C_VEL
LIN {X 0,Y 327.045,Z 340.749,A -85,B 0,C 180,E1 -15032.463,E2 -15032.463} C_VEL
LIN {X 0,Y 326.994,Z 340.754,A -85,B 0,C 180,E1 -15036.169,E2 -15036.169} C_VEL
LIN {X 0,Y 326.912,Z 340.763,A -85,B 0,C 180,E1 -15038.655,E2 -15038.655} C_VEL
LIN {X 0,Y 326.733,Z 340.787,A -85,B 0,C 180,E1 -15042.422,E2 -15042.422} C_VEL
LIN {X 0,Y 326.752,Z 340.781,A -85,B 0,C 180,E1 -15044.958,E2 -15044.958} C_VEL
LIN {X 0,Y 326.731,Z 340.784,A -85,B 0,C 180,E1 -15048.839,E2 -15048.839} C_VEL
LIN {X 0,Y 326.619,Z 340.798,A -85,B 0,C 180,E1 -15052.788,E2 -15052.788} C_VEL
LIN {X 0,Y 326.688,Z 340.789,A -85,B 0,C 180,E1 -15055.484,E2 -15055.484} C_VEL
LIN {X 0,Y 326.646,Z 340.795,A -85,B 0,C 180,E1 -15059.661,E2 -15059.661} C_VEL
LIN {X 0,Y 326.617,Z 340.797,A -85,B 0,C 180,E1 -15062.947,E2 -15062.947} C_VEL
LIN {X 0,Y 326.611,Z 340.799,A -85,B 0,C 180,E1 -15065.52,E2 -15065.52} C_VEL
LIN {X 0,Y 326.611,Z 340.798,A -85,B 0,C 180,E1 -15069.228,E2 -15069.228} C_VEL
LIN {X 0,Y 326.575,Z 340.802,A -85,B 0,C 180,E1 -15072.973,E2 -15072.973} C_VEL
LIN {X 0,Y 326.576,Z 340.802,A -85,B 0,C 180,E1 -15077.029,E2 -15077.029} C_VEL
LIN {X 0,Y 326.612,Z 340.798,A -85,B 0,C 180,E1 -15080.774,E2 -15080.774} C_VEL
LIN {X 0,Y 326.613,Z 340.799,A -85,B 0,C 180,E1 -15084.481,E2 -15084.481} C_VEL
LIN {X 0,Y 326.577,Z 340.8,A -85,B 0,C 180,E1 -15088.07,E2 -15088.07} C_VEL
LIN {X 0,Y 326.722,Z 340.976,A -85,B 0,C 180,E1 -15090.28,E2 -15090.28} C_VEL
LIN {X 0,Y 333.399,Z 361.682,A -85,B 0,C 180,E1 -15091.188,E2 -15091.188} C_VEL
LIN {X 0,Y 333.37,Z 363.605,A -85,B 0,C 180,E1 -15091.243,E2 -15091.243} C_VEL
LIN {X 0,Y 332.592,Z 369.403,A -85,B 0,C 180,E1 -15091.381,E2 -15091.381} C_VEL
LIN {X 0,Y 326.376,Z 388.176,A -85,B 0,C 180,E1 -15091.693,E2 -15091.693} C_VEL
LIN {X 0,Y 325.512,Z 393.98,A -85,B 0,C 180,E1 -15091.83,E2 -15091.83} C_VEL
LIN {X 0,Y 324.747,Z 429.087,A -85,B 0,C 180,E1 -15092.887,E2 -15092.887} C_VEL
LIN {X 0,Y 324.469,Z 441.23,A -85,B 0,C 180,E1 -15093.466,E2 -15093.466} C_VEL
LIN {X 0,Y 323.905,Z 454.763,A -85,B 0,C 180,E1 -15094.368,E2 -15094.368} C_VEL
LIN {X 0,Y 323.339,Z 466.907,A -85,B 0,C 180,E1 -15095.438,E2 -15095.438} C_VEL
LIN {X 0,Y 322.582,Z 478.08,A -85,B 0,C 180,E1 -15096.678,E2 -15096.678} C_VEL
LIN {X 0,Y 321.784,Z 489.176,A -85,B 0,C 180,E1 -15098.205,E2 -15098.205} C_VEL
LIN {X 0,Y 321.109,Z 498.523,A -85,B 0,C 180,E1 -15099.796,E2 -15099.796} C_VEL
LIN {X 0,Y 320.482,Z 506.6,A -85,B 0,C 180,E1 -15101.46,E2 -15101.46} C_VEL
LIN {X 0,Y 319.95,Z 514.255,A -85,B 0,C 180,E1 -15103.408,E2 -15103.408} C_VEL
LIN {X 0,Y 319.563,Z 520.427,A -85,B 0,C 180,E1 -15105.394,E2 -15105.394} C_VEL
LIN {X 0,Y 319.324,Z 525.041,A -85,B 0,C 180,E1 -15107.286,E2 -15107.286} C_VEL
LIN {X 0,Y 319.216,Z 527.549,A -85,B 0,C 180,E1 -15108.572,E2 -15108.572} C_VEL
LIN {X 0,Y 319.23,Z 529.526,A -85,B 0,C 180,E1 -15109.857,E2 -15109.857} C_VEL
LIN {X 0,Y 319.397,Z 531.823,A -85,B 0,C 180,E1 -15111.967,E2 -15111.967} C_VEL
LIN {X 0,Y 319.581,Z 532.798,A -85,B 0,C 180,E1 -15113.688,E2 -15113.688} C_VEL
LIN {X 0,Y 319.697,Z 533.045,A -85,B 0,C 180,E1 -15114.956,E2 -15114.956} C_VEL
LIN {X 0,Y 320.038,Z 532.809,A -85,B 0,C 180,E1 -15116.223,E2 -15116.223} C_VEL
LIN {X 0,Y 320.436,Z 532.135,A -85,B 0,C 180,E1 -15117.486,E2 -15117.486} C_VEL
LIN {X 0,Y 320.915,Z 531.06,A -85,B 0,C 180,E1 -15118.746,E2 -15118.746} C_VEL
LIN {X 0,Y 321.454,Z 529.532,A -85,B 0,C 180,E1 -15120.001,E2 -15120.001} C_VEL
LIN {X 0,Y 322.435,Z 526.375,A -85,B 0,C 180,E1 -15121.874,E2 -15121.874} C_VEL
LIN {X 0,Y 323.676,Z 522.076,A -85,B 0,C 180,E1 -15123.735,E2 -15123.735} C_VEL
LIN {X 0,Y 325.226,Z 515.793,A -85,B 0,C 180,E1 -15125.812,E2 -15125.812} C_VEL
LIN {X 0,Y 326.892,Z 508.633,A -85,B 0,C 180,E1 -15127.645,E2 -15127.645} C_VEL
LIN {X 0,Y 328.505,Z 500.632,A -85,B 0,C 180,E1 -15129.304,E2 -15129.304} C_VEL
LIN {X 0,Y 330.298,Z 491.12,A -85,B 0,C 180,E1 -15130.886,E2 -15130.886} C_VEL
LIN {X 0,Y 331.794,Z 481.13,A -85,B 0,C 180,E1 -15132.229,E2 -15132.229} C_VEL
LIN {X 0,Y 333.285,Z 470.158,A -85,B 0,C 180,E1 -15133.413,E2 -15133.413} C_VEL
LIN {X 0,Y 334.542,Z 458.523,A -85,B 0,C 180,E1 -15134.408,E2 -15134.408} C_VEL
LIN {X 0,Y 335.495,Z 445.611,A -85,B 0,C 180,E1 -15135.258,E2 -15135.258} C_VEL
LIN {X 0,Y 336.064,Z 433.17,A -85,B 0,C 180,E1 -15135.839,E2 -15135.839} C_VEL
LIN {X 0,Y 337.754,Z 402.009,A -85,B 0,C 180,E1 -15136.894,E2 -15136.894} C_VEL
LIN {X 0,Y 339.7,Z 375.511,A -85,B 0,C 180,E1 -15137.772,E2 -15137.772} C_VEL
LIN {X 0,Y 334.666,Z 365.778,A -85,B 0,C 180,E1 -15139.015,E2 -15139.015} C_VEL
LIN {X 0,Y 329.823,Z 357.79,A -85,B 0,C 180,E1 -15140.279,E2 -15140.279} C_VEL
LIN {X 0,Y 327.71,Z 354.564,A -85,B 0,C 180,E1 -15140.858,E2 -15140.858} C_VEL
LIN {X 0,Y 325.445,Z 350.993,A -85,B 0,C 180,E1 -15141.524,E2 -15141.524} C_VEL
LIN {X 0,Y 323.252,Z 347.837,A -85,B 0,C 180,E1 -15142.175,E2 -15142.175} C_VEL
LIN {X 0,Y 322.669,Z 346.688,A -85,B 0,C 180,E1 -15142.369,E2 -15142.369} C_VEL
LIN {X 0,Y 320.551,Z 344.497,A -85,B 0,C 180,E1 -15143.008,E2 -15143.008} C_VEL
LIN {X 0,Y 319.576,Z 341.953,A -85,B 0,C 180,E1 -15143.405,E2 -15143.405} C_VEL
LIN {X 0,Y 319.551,Z 341.68,A -85,B 0,C 180,E1 -15143.493,E2 -15143.493} C_VEL
LIN {X 0,Y 319.554,Z 341.682,A -85,B 0,C 180,E1 -15146.096,E2 -15146.096} C_VEL
LIN {X 0,Y 319.529,Z 341.683,A -85,B 0,C 180,E1 -15148.94,E2 -15148.94} C_VEL
LIN {X 0,Y 319.528,Z 341.682,A -85,B 0,C 180,E1 -15151.863,E2 -15151.863} C_VEL
LIN {X 0,Y 319.582,Z 341.673,A -85,B 0,C 180,E1 -15155.542,E2 -15155.542} C_VEL
LIN {X 0,Y 319.532,Z 341.677,A -85,B 0,C 180,E1 -15159.662,E2 -15159.662} C_VEL
LIN {X 0,Y 319.523,Z 341.682,A -85,B 0,C 180,E1 -15163.46,E2 -15163.46} C_VEL
LIN {X 0,Y 319.555,Z 341.679,A -85,B 0,C 180,E1 -15167.016,E2 -15167.016} C_VEL
LIN {X 0,Y 319.548,Z 341.681,A -85,B 0,C 180,E1 -15170.371,E2 -15170.371} C_VEL
LIN {X 0,Y 319.611,Z 341.674,A -85,B 0,C 180,E1 -15174.693,E2 -15174.693} C_VEL
LIN {X 0,Y 319.641,Z 341.768,A -85,B 0,C 180,E1 -15174.796,E2 -15174.796} C_VEL
LIN {X 0,Y 322.282,Z 351.99,A -85,B 0,C 180,E1 -15176.786,E2 -15176.786} C_VEL
LIN {X 0,Y 325.542,Z 362.117,A -85,B 0,C 180,E1 -15178.58,E2 -15178.58} C_VEL
LIN {X 0,Y 327.982,Z 371.304,A -85,B 0,C 180,E1 -15179.895,E2 -15179.895} C_VEL
LIN {X 0,Y 329.549,Z 382.355,A -85,B 0,C 180,E1 -15180.804,E2 -15180.804} C_VEL
LIN {X 0,Y 331.699,Z 397.808,A -85,B 0,C 180,E1 -15181.907,E2 -15181.907} C_VEL
LIN {X 0,Y 334.063,Z 421.827,A -85,B 0,C 180,E1 -15183.365,E2 -15183.365} C_VEL
LIN {X 0,Y 335.183,Z 439.7,A -85,B 0,C 180,E1 -15184.297,E2 -15184.297} C_VEL
LIN {X 0,Y 335.531,Z 453.868,A -85,B 0,C 180,E1 -15184.932,E2 -15184.932} C_VEL
LIN {X 0,Y 332.632,Z 500.247,A -85,B 0,C 180,E1 -15186.455,E2 -15186.455} C_VEL
LIN {X 0,Y 331.231,Z 514.236,A -85,B 0,C 180,E1 -15187.135,E2 -15187.135} C_VEL
LIN {X 0,Y 329.271,Z 528.195,A -85,B 0,C 180,E1 -15188.067,E2 -15188.067} C_VEL
LIN {X 0,Y 327.357,Z 539.941,A -85,B 0,C 180,E1 -15189.088,E2 -15189.088} C_VEL
LIN {X 0,Y 325.303,Z 551.942,A -85,B 0,C 180,E1 -15190.435,E2 -15190.435} C_VEL
LIN {X 0,Y 323.301,Z 562.84,A -85,B 0,C 180,E1 -15191.954,E2 -15191.954} C_VEL
LIN {X 0,Y 321.678,Z 571.856,A -85,B 0,C 180,E1 -15193.499,E2 -15193.499} C_VEL
LIN {X 0,Y 320.343,Z 580.785,A -85,B 0,C 180,E1 -15195.386,E2 -15195.386} C_VEL
LIN {X 0,Y 319.274,Z 588.1,A -85,B 0,C 180,E1 -15197.283,E2 -15197.283} C_VEL
LIN {X 0,Y 318.615,Z 594.043,A -85,B 0,C 180,E1 -15199.193,E2 -15199.193} C_VEL
LIN {X 0,Y 318.378,Z 598.764,A -85,B 0,C 180,E1 -15201.111,E2 -15201.111} C_VEL
LIN {X 0,Y 318.424,Z 602.81,A -85,B 0,C 180,E1 -15203.321,E2 -15203.321} C_VEL
LIN {X 0,Y 318.567,Z 604.932,A -85,B 0,C 180,E1 -15204.937,E2 -15204.937} C_VEL
LIN {X 0,Y 318.779,Z 606.059,A -85,B 0,C 180,E1 -15206.207,E2 -15206.207} C_VEL
LIN {X 0,Y 319.049,Z 607.122,A -85,B 0,C 180,E1 -15208.738,E2 -15208.738} C_VEL
LIN {X 0,Y 319.073,Z 607.931,A -85,B 0,C 180,E1 -15210,E2 -15210} C_VEL
LIN {X 0,Y 318.909,Z 608.263,A -85,B 0,C 180,E1 -15211.263,E2 -15211.263} C_VEL
LIN {X 0,Y 318.804,Z 608.134,A -85,B 0,C 180,E1 -15212.527,E2 -15212.527} C_VEL
LIN {X 0,Y 318.689,Z 607.515,A -85,B 0,C 180,E1 -15213.793,E2 -15213.793} C_VEL
LIN {X 0,Y 318.462,Z 606.445,A -85,B 0,C 180,E1 -15215.064,E2 -15215.064} C_VEL
LIN {X 0,Y 318.346,Z 604.649,A -85,B 0,C 180,E1 -15216.559,E2 -15216.559} C_VEL
LIN {X 0,Y 318.301,Z 600.555,A -85,B 0,C 180,E1 -15218.891,E2 -15218.891} C_VEL
LIN {X 0,Y 318.557,Z 596.021,A -85,B 0,C 180,E1 -15220.808,E2 -15220.808} C_VEL
LIN {X 0,Y 319.432,Z 589.273,A -85,B 0,C 180,E1 -15223.033,E2 -15223.033} C_VEL
LIN {X 0,Y 320.584,Z 582.055,A -85,B 0,C 180,E1 -15224.927,E2 -15224.927} C_VEL
LIN {X 0,Y 322.059,Z 573.232,A -85,B 0,C 180,E1 -15226.807,E2 -15226.807} C_VEL
LIN {X 0,Y 323.774,Z 564.428,A -85,B 0,C 180,E1 -15228.345,E2 -15228.345} C_VEL
LIN {X 0,Y 325.857,Z 553.937,A -85,B 0,C 180,E1 -15229.858,E2 -15229.858} C_VEL
LIN {X 0,Y 328.068,Z 542.43,A -85,B 0,C 180,E1 -15231.192,E2 -15231.192} C_VEL
LIN {X 0,Y 330.326,Z 529.903,A -85,B 0,C 180,E1 -15232.353,E2 -15232.353} C_VEL
LIN {X 0,Y 332.493,Z 515.889,A -85,B 0,C 180,E1 -15233.348,E2 -15233.348} C_VEL
LIN {X 0,Y 334.205,Z 502.075,A -85,B 0,C 180,E1 -15234.085,E2 -15234.085} C_VEL
LIN {X 0,Y 335.858,Z 481.492,A -85,B 0,C 180,E1 -15234.834,E2 -15234.834} C_VEL
LIN {X 0,Y 337.992,Z 449.827,A -85,B 0,C 180,E1 -15235.945,E2 -15235.945} C_VEL
LIN {X 0,Y 337.575,Z 434.673,A -85,B 0,C 180,E1 -15236.718,E2 -15236.718} C_VEL
LIN {X 0,Y 336.628,Z 421.854,A -85,B 0,C 180,E1 -15237.493,E2 -15237.493} C_VEL
LIN {X 0,Y 334.441,Z 404.789,A -85,B 0,C 180,E1 -15238.751,E2 -15238.751} C_VEL
LIN {X 0,Y 331.845,Z 389.558,A -85,B 0,C 180,E1 -15240.102,E2 -15240.102} C_VEL
LIN {X 0,Y 329.842,Z 379.336,A -85,B 0,C 180,E1 -15241.172,E2 -15241.172} C_VEL
LIN {X 0,Y 328.688,Z 372.232,A -85,B 0,C 180,E1 -15243.498,E2 -15243.498} C_VEL
LIN {X 0,Y 327.096,Z 365.116,A -85,B 0,C 180,E1 -15246.218,E2 -15246.218} C_VEL
LIN {X 0,Y 325.355,Z 359.173,A -85,B 0,C 180,E1 -15248.955,E2 -15248.955} C_VEL
LIN {X 0,Y 323.503,Z 353.265,A -85,B 0,C 180,E1 -15252.384,E2 -15252.384} C_VEL
LIN {X 0,Y 322.049,Z 349.126,A -85,B 0,C 180,E1 -15255.706,E2 -15255.706} C_VEL
LIN {X 0,Y 321.062,Z 346.467,A -85,B 0,C 180,E1 -15258.951,E2 -15258.951} C_VEL
LIN {X 0,Y 320.653,Z 345.021,A -85,B 0,C 180,E1 -15262.142,E2 -15262.142} C_VEL
LIN {X 0,Y 320.599,Z 344.757,A -85,B 0,C 180,E1 -15265.252,E2 -15265.252} C_VEL
LIN {X 0,Y 320.808,Z 345.798,A -85,B 0,C 180,E1 -15268.509,E2 -15268.509} C_VEL
LIN {X 0,Y 323.459,Z 348.767,A -85,B 0,C 180,E1 -15269.663,E2 -15269.663} C_VEL
LIN {X 0,Y 324.773,Z 349.883,A -85,B 0,C 180,E1 -15270.151,E2 -15270.151} C_VEL
LIN {X 0,Y 327.415,Z 353.218,A -85,B 0,C 180,E1 -15271.154,E2 -15271.154} C_VEL
LIN {X 0,Y 329.961,Z 356.709,A -85,B 0,C 180,E1 -15272.057,E2 -15272.057} C_VEL
LIN {X 0,Y 333.92,Z 363.114,A -85,B 0,C 180,E1 -15273.38,E2 -15273.38} C_VEL
LIN {X 0,Y 337.226,Z 368.503,A -85,B 0,C 180,E1 -15274.382,E2 -15274.382} C_VEL
LIN {X 0,Y 342.086,Z 377.858,A -85,B 0,C 180,E1 -15275.782,E2 -15275.782} C_VEL
LIN {X 0,Y 338.009,Z 428.603,A -85,B 0,C 180,E1 -15277.619,E2 -15277.619} C_VEL
LIN {X 0,Y 337.259,Z 443.902,A -85,B 0,C 180,E1 -15278.291,E2 -15278.291} C_VEL
LIN {X 0,Y 336.232,Z 456.905,A -85,B 0,C 180,E1 -15279.105,E2 -15279.105} C_VEL
LIN {X 0,Y 334.96,Z 468.679,A -85,B 0,C 180,E1 -15280.065,E2 -15280.065} C_VEL
LIN {X 0,Y 333.399,Z 480.02,A -85,B 0,C 180,E1 -15281.248,E2 -15281.248} C_VEL
LIN {X 0,Y 331.69,Z 490.272,A -85,B 0,C 180,E1 -15282.569,E2 -15282.569} C_VEL
LIN {X 0,Y 330.078,Z 498.868,A -85,B 0,C 180,E1 -15283.93,E2 -15283.93} C_VEL
LIN {X 0,Y 328.411,Z 506.74,A -85,B 0,C 180,E1 -15285.436,E2 -15285.436} C_VEL
LIN {X 0,Y 326.568,Z 514.398,A -85,B 0,C 180,E1 -15287.256,E2 -15287.256} C_VEL
LIN {X 0,Y 325.195,Z 519.627,A -85,B 0,C 180,E1 -15288.784,E2 -15288.784} C_VEL
LIN {X 0,Y 323.753,Z 524.652,A -85,B 0,C 180,E1 -15290.629,E2 -15290.629} C_VEL
LIN {X 0,Y 322.503,Z 528.52,A -85,B 0,C 180,E1 -15292.486,E2 -15292.486} C_VEL
LIN {X 0,Y 321.829,Z 530.495,A -85,B 0,C 180,E1 -15293.731,E2 -15293.731} C_VEL
LIN {X 0,Y 321.194,Z 532.001,A -85,B 0,C 180,E1 -15294.978,E2 -15294.978} C_VEL
LIN {X 0,Y 320.707,Z 533.049,A -85,B 0,C 180,E1 -15296.23,E2 -15296.23} C_VEL
LIN {X 0,Y 320.321,Z 533.684,A -85,B 0,C 180,E1 -15297.484,E2 -15297.484} C_VEL
LIN {X 0,Y 319.932,Z 533.906,A -85,B 0,C 180,E1 -15298.741,E2 -15298.741} C_VEL
LIN {X 0,Y 319.78,Z 533.643,A -85,B 0,C 180,E1 -15299.999,E2 -15299.999} C_VEL
LIN {X 0,Y 319.421,Z 533.007,A -85,B 0,C 180,E1 -15301.26,E2 -15301.26} C_VEL
LIN {X 0,Y 319.05,Z 531.963,A -85,B 0,C 180,E1 -15302.524,E2 -15302.524} C_VEL
LIN {X 0,Y 319.15,Z 530.401,A -85,B 0,C 180,E1 -15303.787,E2 -15303.787} C_VEL
LIN {X 0,Y 319.369,Z 527.249,A -85,B 0,C 180,E1 -15305.682,E2 -15305.682} C_VEL
LIN {X 0,Y 319.416,Z 523.016,A -85,B 0,C 180,E1 -15307.585,E2 -15307.585} C_VEL
LIN {X 0,Y 319.755,Z 516.545,A -85,B 0,C 180,E1 -15309.807,E2 -15309.807} C_VEL
LIN {X 0,Y 320.191,Z 509.433,A -85,B 0,C 180,E1 -15311.714,E2 -15311.714} C_VEL
LIN {X 0,Y 320.798,Z 500.609,A -85,B 0,C 180,E1 -15313.621,E2 -15313.621} C_VEL
LIN {X 0,Y 321.4,Z 491.599,A -85,B 0,C 180,E1 -15315.212,E2 -15315.212} C_VEL
LIN {X 0,Y 322.154,Z 480.478,A -85,B 0,C 180,E1 -15316.801,E2 -15316.801} C_VEL
LIN {X 0,Y 322.832,Z 469.537,A -85,B 0,C 180,E1 -15318.072,E2 -15318.072} C_VEL
LIN {X 0,Y 323.403,Z 457.489,A -85,B 0,C 180,E1 -15319.188,E2 -15319.188} C_VEL
LIN {X 0,Y 324.074,Z 444.156,A -85,B 0,C 180,E1 -15320.137,E2 -15320.137} C_VEL
LIN {X 0,Y 324.353,Z 430.57,A -85,B 0,C 180,E1 -15320.834,E2 -15320.834} C_VEL
LIN {X 0,Y 324.804,Z 406.344,A -85,B 0,C 180,E1 -15321.622,E2 -15321.622} C_VEL
LIN {X 0,Y 326.009,Z 362.036,A -85,B 0,C 180,E1 -15322.967,E2 -15322.967} C_VEL
LIN {X 0,Y 319.656,Z 341.664,A -85,B 0,C 180,E1 -15323.915,E2 -15323.915} C_VEL
LIN {X 0,Y 319.608,Z 341.671,A -85,B 0,C 180,E1 -15327.501,E2 -15327.501} C_VEL
LIN {X 0,Y 319.57,Z 341.68,A -85,B 0,C 180,E1 -15330.941,E2 -15330.941} C_VEL
LIN {X 0,Y 319.559,Z 341.681,A -85,B 0,C 180,E1 -15334.876,E2 -15334.876} C_VEL
LIN {X 0,Y 319.541,Z 341.678,A -85,B 0,C 180,E1 -15338.012,E2 -15338.012} C_VEL
LIN {X 0,Y 319.524,Z 341.681,A -85,B 0,C 180,E1 -15341.597,E2 -15341.597} C_VEL
LIN {X 0,Y 319.513,Z 341.688,A -85,B 0,C 180,E1 -15344.737,E2 -15344.737} C_VEL
LIN {X 0,Y 319.524,Z 341.683,A -85,B 0,C 180,E1 -15348.402,E2 -15348.402} C_VEL
LIN {X 0,Y 319.576,Z 341.677,A -85,B 0,C 180,E1 -15352.343,E2 -15352.343} C_VEL
LIN {X 0,Y 319.558,Z 341.678,A -85,B 0,C 180,E1 -15355.123,E2 -15355.123} C_VEL
LIN {X 0,Y 319.563,Z 341.678,A -85,B 0,C 180,E1 -15359.059,E2 -15359.059} C_VEL
LIN {X 0,Y 319.603,Z 341.675,A -85,B 0,C 180,E1 -15362.498,E2 -15362.498} C_VEL
LIN {X 0,Y 319.602,Z 341.671,A -85,B 0,C 180,E1 -15365.304,E2 -15365.304} C_VEL
LIN {X 0,Y 319.595,Z 341.673,A -85,B 0,C 180,E1 -15368.048,E2 -15368.048} C_VEL
LIN {X 0,Y 319.686,Z 341.662,A -85,B 0,C 180,E1 -15370.962,E2 -15370.962} C_VEL
LIN {X 0,Y 319.728,Z 341.655,A -85,B 0,C 180,E1 -15375.276,E2 -15375.276} C_VEL
LIN {X 0,Y 319.755,Z 341.653,A -85,B 0,C 180,E1 -15379.873,E2 -15379.873} C_VEL
LIN {X 0,Y 319.931,Z 341.635,A -85,B 0,C 180,E1 -15382.426,E2 -15382.426} C_VEL
LIN {X 0,Y 319.745,Z 341.654,A -85,B 0,C 180,E1 -15384.956,E2 -15384.956} C_VEL
LIN {X 0,Y 319.989,Z 341.623,A -85,B 0,C 180,E1 -15387.483,E2 -15387.483} C_VEL
LIN {X 0,Y 320.148,Z 341.605,A -85,B 0,C 180,E1 -15390,E2 -15390} C_VEL
LIN {X 0,Y 319.989,Z 341.627,A -85,B 0,C 180,E1 -15392.518,E2 -15392.518} C_VEL
LIN {X 0,Y 319.949,Z 341.633,A -85,B 0,C 180,E1 -15396.306,E2 -15396.306} C_VEL
LIN {X 0,Y 319.84,Z 341.642,A -85,B 0,C 180,E1 -15398.848,E2 -15398.848} C_VEL
LIN {X 0,Y 319.68,Z 341.663,A -85,B 0,C 180,E1 -15402.7,E2 -15402.7} C_VEL
LIN {X 0,Y 319.697,Z 341.659,A -85,B 0,C 180,E1 -15405.296,E2 -15405.296} C_VEL
LIN {X 0,Y 319.673,Z 341.662,A -85,B 0,C 180,E1 -15409.255,E2 -15409.255} C_VEL
LIN {X 0,Y 319.568,Z 341.675,A -85,B 0,C 180,E1 -15413.32,E2 -15413.32} C_VEL
LIN {X 0,Y 319.632,Z 341.672,A -85,B 0,C 180,E1 -15416.089,E2 -15416.089} C_VEL
LIN {X 0,Y 319.578,Z 341.674,A -85,B 0,C 180,E1 -15418.935,E2 -15418.935} C_VEL
LIN {X 0,Y 319.53,Z 341.683,A -85,B 0,C 180,E1 -15421.862,E2 -15421.862} C_VEL
LIN {X 0,Y 319.579,Z 341.675,A -85,B 0,C 180,E1 -15425.544,E2 -15425.544} C_VEL
LIN {X 0,Y 319.572,Z 341.679,A -85,B 0,C 180,E1 -15428.009,E2 -15428.009} C_VEL
LIN {X 0,Y 319.525,Z 341.682,A -85,B 0,C 180,E1 -15431.598,E2 -15431.598} C_VEL
LIN {X 0,Y 319.488,Z 341.685,A -85,B 0,C 180,E1 -15435.258,E2 -15435.258} C_VEL
LIN {X 0,Y 319.528,Z 341.68,A -85,B 0,C 180,E1 -15438.713,E2 -15438.713} C_VEL
LIN {X 0,Y 319.577,Z 341.676,A -85,B 0,C 180,E1 -15442.345,E2 -15442.345} C_VEL
LIN {X 0,Y 319.56,Z 341.676,A -85,B 0,C 180,E1 -15445.124,E2 -15445.124} C_VEL
LIN {X 0,Y 319.571,Z 341.675,A -85,B 0,C 180,E1 -15449.059,E2 -15449.059} C_VEL
LIN {X 0,Y 319.639,Z 341.672,A -85,B 0,C 180,E1 -15449.966,E2 -15449.966} C_VEL
LIN {X 0,Y 326.446,Z 362.543,A -85,B 0,C 180,E1 -15450.922,E2 -15450.922} C_VEL
LIN {X 0,Y 325.512,Z 393.98,A -85,B 0,C 180,E1 -15451.83,E2 -15451.83} C_VEL
LIN {X 0,Y 324.664,Z 399.782,A -85,B 0,C 180,E1 -15451.967,E2 -15451.967} C_VEL
LIN {X 0,Y 318.594,Z 418.566,A -85,B 0,C 180,E1 -15452.308,E2 -15452.308} C_VEL
LIN {X 0,Y 317.848,Z 424.354,A -85,B 0,C 180,E1 -15452.465,E2 -15452.465} C_VEL
LIN {X 0,Y 317.585,Z 438.442,A -85,B 0,C 180,E1 -15453.067,E2 -15453.067} C_VEL
LIN {X 0,Y 317.14,Z 451.411,A -85,B 0,C 180,E1 -15453.869,E2 -15453.869} C_VEL
LIN {X 0,Y 316.537,Z 463.564,A -85,B 0,C 180,E1 -15454.874,E2 -15454.874} C_VEL
LIN {X 0,Y 315.755,Z 476.122,A -85,B 0,C 180,E1 -15456.202,E2 -15456.202} C_VEL
LIN {X 0,Y 314.972,Z 487.341,A -85,B 0,C 180,E1 -15457.709,E2 -15457.709} C_VEL
LIN {X 0,Y 314.178,Z 497.522,A -85,B 0,C 180,E1 -15459.388,E2 -15459.388} C_VEL
LIN {X 0,Y 313.425,Z 507.106,A -85,B 0,C 180,E1 -15461.366,E2 -15461.366} C_VEL
LIN {X 0,Y 312.866,Z 514.856,A -85,B 0,C 180,E1 -15463.358,E2 -15463.358} C_VEL
LIN {X 0,Y 312.445,Z 521.89,A -85,B 0,C 180,E1 -15465.675,E2 -15465.675} C_VEL
LIN {X 0,Y 312.227,Z 526.499,A -85,B 0,C 180,E1 -15467.653,E2 -15467.653} C_VEL
LIN {X 0,Y 312.155,Z 529.923,A -85,B 0,C 180,E1 -15469.624,E2 -15469.624} C_VEL
LIN {X 0,Y 312.337,Z 532.554,A -85,B 0,C 180,E1 -15471.919,E2 -15471.919} C_VEL
LIN {X 0,Y 312.522,Z 533.626,A -85,B 0,C 180,E1 -15473.545,E2 -15473.545} C_VEL
LIN {X 0,Y 312.644,Z 533.981,A -85,B 0,C 180,E1 -15474.842,E2 -15474.842} C_VEL
LIN {X 0,Y 312.993,Z 533.91,A -85,B 0,C 180,E1 -15476.138,E2 -15476.138} C_VEL
LIN {X 0,Y 313.411,Z 533.407,A -85,B 0,C 180,E1 -15477.43,E2 -15477.43} C_VEL
LIN {X 0,Y 313.902,Z 532.443,A -85,B 0,C 180,E1 -15478.718,E2 -15478.718} C_VEL
LIN {X 0,Y 314.463,Z 531.073,A -85,B 0,C 180,E1 -15480.001,E2 -15480.001} C_VEL
LIN {X 0,Y 315.515,Z 528.138,A -85,B 0,C 180,E1 -15481.915,E2 -15481.915} C_VEL
LIN {X 0,Y 316.775,Z 524.105,A -85,B 0,C 180,E1 -15483.817,E2 -15483.817} C_VEL
LIN {X 0,Y 318.228,Z 518.899,A -85,B 0,C 180,E1 -15485.704,E2 -15485.704} C_VEL
LIN {X 0,Y 319.895,Z 512.303,A -85,B 0,C 180,E1 -15487.575,E2 -15487.575} C_VEL
LIN {X 0,Y 321.81,Z 504.078,A -85,B 0,C 180,E1 -15489.428,E2 -15489.428} C_VEL
LIN {X 0,Y 323.47,Z 495.626,A -85,B 0,C 180,E1 -15490.96,E2 -15490.96} C_VEL
LIN {X 0,Y 325.329,Z 485.35,A -85,B 0,C 180,E1 -15492.476,E2 -15492.476} C_VEL
LIN {X 0,Y 326.897,Z 475.231,A -85,B 0,C 180,E1 -15493.68,E2 -15493.68} C_VEL
LIN {X 0,Y 328.386,Z 463.465,A -85,B 0,C 180,E1 -15494.783,E2 -15494.783} C_VEL
LIN {X 0,Y 329.495,Z 450.842,A -85,B 0,C 180,E1 -15495.711,E2 -15495.711} C_VEL
LIN {X 0,Y 330.276,Z 437.606,A -85,B 0,C 180,E1 -15496.417,E2 -15496.417} C_VEL
LIN {X 0,Y 331.832,Z 409.651,A -85,B 0,C 180,E1 -15497.433,E2 -15497.433} C_VEL
LIN {X 0,Y 334.226,Z 378.111,A -85,B 0,C 180,E1 -15498.504,E2 -15498.504} C_VEL
LIN {X 0,Y 328.822,Z 367.734,A -85,B 0,C 180,E1 -15499.953,E2 -15499.953} C_VEL
LIN {X 0,Y 323.741,Z 359.679,A -85,B 0,C 180,E1 -15501.39,E2 -15501.39} C_VEL
LIN {X 0,Y 321.658,Z 356.44,A -85,B 0,C 180,E1 -15502.019,E2 -15502.019} C_VEL
LIN {X 0,Y 319.09,Z 352.425,A -85,B 0,C 180,E1 -15502.859,E2 -15502.859} C_VEL
LIN {X 0,Y 316.876,Z 349.681,A -85,B 0,C 180,E1 -15503.583,E2 -15503.583} C_VEL
LIN {X 0,Y 315.758,Z 347.662,A -85,B 0,C 180,E1 -15503.999,E2 -15503.999} C_VEL
LIN {X 0,Y 313.558,Z 345.495,A -85,B 0,C 180,E1 -15504.759,E2 -15504.759} C_VEL
LIN {X 0,Y 312.557,Z 342.919,A -85,B 0,C 180,E1 -15505.232,E2 -15505.232} C_VEL
LIN {X 0,Y 312.517,Z 342.56,A -85,B 0,C 180,E1 -15505.296,E2 -15505.296} C_VEL
LIN {X 0,Y 312.489,Z 342.56,A -85,B 0,C 180,E1 -15508.701,E2 -15508.701} C_VEL
LIN {X 0,Y 312.505,Z 342.558,A -85,B 0,C 180,E1 -15512.667,E2 -15512.667} C_VEL
LIN {X 0,Y 312.537,Z 342.551,A -85,B 0,C 180,E1 -15515.949,E2 -15515.949} C_VEL
LIN {X 0,Y 312.458,Z 342.559,A -85,B 0,C 180,E1 -15520.115,E2 -15520.115} C_VEL
LIN {X 0,Y 312.46,Z 342.561,A -85,B 0,C 180,E1 -15523.965,E2 -15523.965} C_VEL
LIN {X 0,Y 312.459,Z 342.566,A -85,B 0,C 180,E1 -15527.925,E2 -15527.925} C_VEL
LIN {X 0,Y 312.488,Z 342.561,A -85,B 0,C 180,E1 -15531.922,E2 -15531.922} C_VEL
LIN {X 0,Y 312.495,Z 342.56,A -85,B 0,C 180,E1 -15532.706,E2 -15532.706} C_VEL
LIN {X 0,Y 312.965,Z 344.344,A -85,B 0,C 180,E1 -15533.16,E2 -15533.16} C_VEL
LIN {X 0,Y 315.852,Z 348.357,A -85,B 0,C 180,E1 -15534.653,E2 -15534.653} C_VEL
LIN {X 0,Y 319.6,Z 362.72,A -85,B 0,C 180,E1 -15537.374,E2 -15537.374} C_VEL
LIN {X 0,Y 321.241,Z 368.415,A -85,B 0,C 180,E1 -15538.327,E2 -15538.327} C_VEL
LIN {X 0,Y 323.32,Z 375.667,A -85,B 0,C 180,E1 -15539.283,E2 -15539.283} C_VEL
LIN {X 0,Y 325.551,Z 391.959,A -85,B 0,C 180,E1 -15540.564,E2 -15540.564} C_VEL
LIN {X 0,Y 327.364,Z 408.561,A -85,B 0,C 180,E1 -15541.713,E2 -15541.713} C_VEL
LIN {X 0,Y 329.126,Z 430.096,A -85,B 0,C 180,E1 -15543.015,E2 -15543.015} C_VEL
LIN {X 0,Y 329.968,Z 452.656,A -85,B 0,C 180,E1 -15544.134,E2 -15544.134} C_VEL
LIN {X 0,Y 326.74,Z 500.015,A -85,B 0,C 180,E1 -15545.751,E2 -15545.751} C_VEL
LIN {X 0,Y 325.315,Z 513.668,A -85,B 0,C 180,E1 -15546.442,E2 -15546.442} C_VEL
LIN {X 0,Y 323.392,Z 526.435,A -85,B 0,C 180,E1 -15547.31,E2 -15547.31} C_VEL
LIN {X 0,Y 321.363,Z 538.188,A -85,B 0,C 180,E1 -15548.343,E2 -15548.343} C_VEL
LIN {X 0,Y 319.112,Z 550.286,A -85,B 0,C 180,E1 -15549.704,E2 -15549.704} C_VEL
LIN {X 0,Y 317.013,Z 561.296,A -85,B 0,C 180,E1 -15551.249,E2 -15551.249} C_VEL
LIN {X 0,Y 315.177,Z 570.359,A -85,B 0,C 180,E1 -15552.815,E2 -15552.815} C_VEL
LIN {X 0,Y 313.677,Z 578.976,A -85,B 0,C 180,E1 -15554.653,E2 -15554.653} C_VEL
LIN {X 0,Y 312.468,Z 586.717,A -85,B 0,C 180,E1 -15556.671,E2 -15556.671} C_VEL
LIN {X 0,Y 311.572,Z 593.578,A -85,B 0,C 180,E1 -15558.946,E2 -15558.946} C_VEL
LIN {X 0,Y 311.286,Z 598.158,A -85,B 0,C 180,E1 -15560.907,E2 -15560.907} C_VEL
LIN {X 0,Y 311.357,Z 602.314,A -85,B 0,C 180,E1 -15563.307,E2 -15563.307} C_VEL
LIN {X 0,Y 311.48,Z 604.136,A -85,B 0,C 180,E1 -15564.822,E2 -15564.822} C_VEL
LIN {X 0,Y 311.703,Z 605.21,A -85,B 0,C 180,E1 -15566.121,E2 -15566.121} C_VEL
LIN {X 0,Y 311.859,Z 605.846,A -85,B 0,C 180,E1 -15567.416,E2 -15567.416} C_VEL
LIN {X 0,Y 312.025,Z 606.019,A -85,B 0,C 180,E1 -15568.709,E2 -15568.709} C_VEL
LIN {X 0,Y 312.053,Z 606.844,A -85,B 0,C 180,E1 -15570,E2 -15570} C_VEL
LIN {X 0,Y 311.879,Z 607.227,A -85,B 0,C 180,E1 -15571.291,E2 -15571.291} C_VEL
LIN {X 0,Y 311.754,Z 607.172,A -85,B 0,C 180,E1 -15572.584,E2 -15572.584} C_VEL
LIN {X 0,Y 311.617,Z 606.646,A -85,B 0,C 180,E1 -15573.879,E2 -15573.879} C_VEL
LIN {X 0,Y 311.379,Z 605.631,A -85,B 0,C 180,E1 -15575.18,E2 -15575.18} C_VEL
LIN {X 0,Y 311.265,Z 604.113,A -85,B 0,C 180,E1 -15576.548,E2 -15576.548} C_VEL
LIN {X 0,Y 311.197,Z 601.203,A -85,B 0,C 180,E1 -15578.441,E2 -15578.441} C_VEL
LIN {X 0,Y 311.381,Z 597.16,A -85,B 0,C 180,E1 -15580.402,E2 -15580.402} C_VEL
LIN {X 0,Y 312.026,Z 592.031,A -85,B 0,C 180,E1 -15582.355,E2 -15582.355} C_VEL
LIN {X 0,Y 313.245,Z 584.553,A -85,B 0,C 180,E1 -15584.609,E2 -15584.609} C_VEL
LIN {X 0,Y 314.647,Z 576.632,A -85,B 0,C 180,E1 -15586.513,E2 -15586.513} C_VEL
LIN {X 0,Y 316.673,Z 566.759,A -85,B 0,C 180,E1 -15588.436,E2 -15588.436} C_VEL
LIN {X 0,Y 319.034,Z 555.9,A -85,B 0,C 180,E1 -15590.133,E2 -15590.133} C_VEL
LIN {X 0,Y 321.539,Z 543.814,A -85,B 0,C 180,E1 -15591.644,E2 -15591.644} C_VEL
LIN {X 0,Y 323.844,Z 531.995,A -85,B 0,C 180,E1 -15592.825,E2 -15592.825} C_VEL
LIN {X 0,Y 326.31,Z 517.979,A -85,B 0,C 180,E1 -15593.902,E2 -15593.902} C_VEL
LIN {X 0,Y 328.207,Z 503.997,A -85,B 0,C 180,E1 -15594.723,E2 -15594.723} C_VEL
LIN {X 0,Y 329.752,Z 489.146,A -85,B 0,C 180,E1 -15595.332,E2 -15595.332} C_VEL
LIN {X 0,Y 332.576,Z 450.971,A -85,B 0,C 180,E1 -15596.701,E2 -15596.701} C_VEL
LIN {X 0,Y 332.26,Z 435.311,A -85,B 0,C 180,E1 -15597.534,E2 -15597.534} C_VEL
LIN {X 0,Y 331.453,Z 423.531,A -85,B 0,C 180,E1 -15598.286,E2 -15598.286} C_VEL
LIN {X 0,Y 329.571,Z 407.33,A -85,B 0,C 180,E1 -15599.53,E2 -15599.53} C_VEL
LIN {X 0,Y 327.158,Z 392.118,A -85,B 0,C 180,E1 -15600.944,E2 -15600.944} C_VEL
LIN {X 0,Y 325.454,Z 383.465,A -85,B 0,C 180,E1 -15601.893,E2 -15601.893} C_VEL
LIN {X 0,Y 322.599,Z 376.62,A -85,B 0,C 180,E1 -15603.144,E2 -15603.144} C_VEL
LIN {X 0,Y 321.094,Z 369.356,A -85,B 0,C 180,E1 -15605.918,E2 -15605.918} C_VEL
LIN {X 0,Y 319.193,Z 362.589,A -85,B 0,C 180,E1 -15609.079,E2 -15609.079} C_VEL
LIN {X 0,Y 317.626,Z 357.554,A -85,B 0,C 180,E1 -15612.026,E2 -15612.026} C_VEL
LIN {X 0,Y 316.408,Z 354.042,A -85,B 0,C 180,E1 -15614.701,E2 -15614.701} C_VEL
LIN {X 0,Y 315.345,Z 350.87,A -85,B 0,C 180,E1 -15618.04,E2 -15618.04} C_VEL
LIN {X 0,Y 314.662,Z 349.071,A -85,B 0,C 180,E1 -15621.419,E2 -15621.419} C_VEL
LIN {X 0,Y 314.597,Z 348.491,A -85,B 0,C 180,E1 -15624.49,E2 -15624.49} C_VEL
LIN {X 0,Y 314.658,Z 348.787,A -85,B 0,C 180,E1 -15626.33,E2 -15626.33} C_VEL
LIN {X 0,Y 317.197,Z 351.625,A -85,B 0,C 180,E1 -15627.731,E2 -15627.731} C_VEL
LIN {X 0,Y 318.628,Z 352.763,A -85,B 0,C 180,E1 -15628.379,E2 -15628.379} C_VEL
LIN {X 0,Y 321.271,Z 355.461,A -85,B 0,C 180,E1 -15629.527,E2 -15629.527} C_VEL
LIN {X 0,Y 324.179,Z 358.933,A -85,B 0,C 180,E1 -15630.688,E2 -15630.688} C_VEL
LIN {X 0,Y 327.434,Z 363.954,A -85,B 0,C 180,E1 -15631.922,E2 -15631.922} C_VEL
LIN {X 0,Y 331.613,Z 370.635,A -85,B 0,C 180,E1 -15633.343,E2 -15633.343} C_VEL
LIN {X 0,Y 336.388,Z 379.732,A -85,B 0,C 180,E1 -15634.855,E2 -15634.855} C_VEL
LIN {X 0,Y 336.987,Z 381.047,A -85,B 0,C 180,E1 -15635.039,E2 -15635.039} C_VEL
LIN {X 0,Y 332.77,Z 428.566,A -85,B 0,C 180,E1 -15636.795,E2 -15636.795} C_VEL
LIN {X 0,Y 331.86,Z 444.533,A -85,B 0,C 180,E1 -15637.51,E2 -15637.51} C_VEL
LIN {X 0,Y 330.757,Z 457.584,A -85,B 0,C 180,E1 -15638.334,E2 -15638.334} C_VEL
LIN {X 0,Y 329.273,Z 470.155,A -85,B 0,C 180,E1 -15639.379,E2 -15639.379} C_VEL
LIN {X 0,Y 327.616,Z 481.351,A -85,B 0,C 180,E1 -15640.579,E2 -15640.579} C_VEL
LIN {X 0,Y 325.756,Z 491.618,A -85,B 0,C 180,E1 -15641.932,E2 -15641.932} C_VEL
LIN {X 0,Y 324.032,Z 500.057,A -85,B 0,C 180,E1 -15643.298,E2 -15643.298} C_VEL
LIN {X 0,Y 322.254,Z 507.885,A -85,B 0,C 180,E1 -15644.828,E2 -15644.828} C_VEL
LIN {X 0,Y 320.26,Z 515.513,A -85,B 0,C 180,E1 -15646.678,E2 -15646.678} C_VEL
LIN {X 0,Y 318.495,Z 521.646,A -85,B 0,C 180,E1 -15648.545,E2 -15648.545} C_VEL
LIN {X 0,Y 316.977,Z 526.462,A -85,B 0,C 180,E1 -15650.427,E2 -15650.427} C_VEL
LIN {X 0,Y 315.656,Z 530.129,A -85,B 0,C 180,E1 -15652.322,E2 -15652.322} C_VEL
LIN {X 0,Y 314.946,Z 531.958,A -85,B 0,C 180,E1 -15653.593,E2 -15653.593} C_VEL
LIN {X 0,Y 314.269,Z 533.342,A -85,B 0,C 180,E1 -15654.867,E2 -15654.867} C_VEL
LIN {X 0,Y 313.742,Z 534.298,A -85,B 0,C 180,E1 -15656.146,E2 -15656.146} C_VEL
LIN {X 0,Y 313.323,Z 534.823,A -85,B 0,C 180,E1 -15657.428,E2 -15657.428} C_VEL
LIN {X 0,Y 312.911,Z 534.9,A -85,B 0,C 180,E1 -15658.712,E2 -15658.712} C_VEL
LIN {X 0,Y 312.751,Z 534.546,A -85,B 0,C 180,E1 -15659.999,E2 -15659.999} C_VEL
LIN {X 0,Y 312.354,Z 533.821,A -85,B 0,C 180,E1 -15661.289,E2 -15661.289} C_VEL
LIN {X 0,Y 311.998,Z 532.623,A -85,B 0,C 180,E1 -15662.582,E2 -15662.582} C_VEL
LIN {X 0,Y 312.149,Z 529.975,A -85,B 0,C 180,E1 -15664.519,E2 -15664.519} C_VEL
LIN {X 0,Y 312.296,Z 526.289,A -85,B 0,C 180,E1 -15666.46,E2 -15666.46} C_VEL
LIN {X 0,Y 312.401,Z 521.455,A -85,B 0,C 180,E1 -15668.41,E2 -15668.41} C_VEL
LIN {X 0,Y 312.782,Z 515.345,A -85,B 0,C 180,E1 -15670.355,E2 -15670.355} C_VEL
LIN {X 0,Y 313.277,Z 507.742,A -85,B 0,C 180,E1 -15672.305,E2 -15672.305} C_VEL
LIN {X 0,Y 313.963,Z 498.217,A -85,B 0,C 180,E1 -15674.254,E2 -15674.254} C_VEL
LIN {X 0,Y 314.608,Z 487.902,A -85,B 0,C 180,E1 -15675.969,E2 -15675.969} C_VEL
LIN {X 0,Y 315.357,Z 476.348,A -85,B 0,C 180,E1 -15677.509,E2 -15677.509} C_VEL
LIN {X 0,Y 316.095,Z 464.166,A -85,B 0,C 180,E1 -15678.807,E2 -15678.807} C_VEL
LIN {X 0,Y 316.819,Z 450.364,A -85,B 0,C 180,E1 -15679.941,E2 -15679.941} C_VEL
LIN {X 0,Y 317.283,Z 436.857,A -85,B 0,C 180,E1 -15680.757,E2 -15680.757} C_VEL
LIN {X 0,Y 317.509,Z 422.937,A -85,B 0,C 180,E1 -15681.333,E2 -15681.333} C_VEL
LIN {X 0,Y 319.104,Z 363.537,A -85,B 0,C 180,E1 -15683.191,E2 -15683.191} C_VEL
LIN {X 0,Y 312.601,Z 342.544,A -85,B 0,C 180,E1 -15684.187,E2 -15684.187} C_VEL
LIN {X 0,Y 312.583,Z 342.549,A -85,B 0,C 180,E1 -15686.722,E2 -15686.722} C_VEL
LIN {X 0,Y 312.545,Z 342.55,A -85,B 0,C 180,E1 -15689.649,E2 -15689.649} C_VEL
LIN {X 0,Y 312.518,Z 342.553,A -85,B 0,C 180,E1 -15693.688,E2 -15693.688} C_VEL
LIN {X 0,Y 312.518,Z 342.554,A -85,B 0,C 180,E1 -15697.385,E2 -15697.385} C_VEL
LIN {X 0,Y 312.488,Z 342.562,A -85,B 0,C 180,E1 -15700.709,E2 -15700.709} C_VEL
LIN {X 0,Y 312.471,Z 342.56,A -85,B 0,C 180,E1 -15704.205,E2 -15704.205} C_VEL
LIN {X 0,Y 312.483,Z 342.558,A -85,B 0,C 180,E1 -15707.918,E2 -15707.918} C_VEL
LIN {X 0,Y 312.533,Z 342.552,A -85,B 0,C 180,E1 -15711.91,E2 -15711.91} C_VEL
LIN {X 0,Y 312.504,Z 342.555,A -85,B 0,C 180,E1 -15715.79,E2 -15715.79} C_VEL
LIN {X 0,Y 312.517,Z 342.557,A -85,B 0,C 180,E1 -15718.853,E2 -15718.853} C_VEL
LIN {X 0,Y 312.567,Z 342.547,A -85,B 0,C 180,E1 -15721.824,E2 -15721.824} C_VEL
LIN {X 0,Y 312.582,Z 342.55,A -85,B 0,C 180,E1 -15724.711,E2 -15724.711} C_VEL
LIN {X 0,Y 312.585,Z 342.545,A -85,B 0,C 180,E1 -15727.529,E2 -15727.529} C_VEL
LIN {X 0,Y 312.635,Z 342.539,A -85,B 0,C 180,E1 -15731.656,E2 -15731.656} C_VEL
LIN {X 0,Y 312.691,Z 342.532,A -85,B 0,C 180,E1 -15735.686,E2 -15735.686} C_VEL
LIN {X 0,Y 312.7,Z 342.531,A -85,B 0,C 180,E1 -15739.642,E2 -15739.642} C_VEL
LIN {X 0,Y 312.869,Z 342.513,A -85,B 0,C 180,E1 -15742.254,E2 -15742.254} C_VEL
LIN {X 0,Y 312.715,Z 342.531,A -85,B 0,C 180,E1 -15744.843,E2 -15744.843} C_VEL
LIN {X 0,Y 312.988,Z 342.497,A -85,B 0,C 180,E1 -15748.714,E2 -15748.714} C_VEL
LIN {X 0,Y 312.988,Z 342.495,A -85,B 0,C 180,E1 -15751.287,E2 -15751.287} C_VEL
LIN {X 0,Y 312.716,Z 342.529,A -85,B 0,C 180,E1 -15755.158,E2 -15755.158} C_VEL
LIN {X 0,Y 312.869,Z 342.51,A -85,B 0,C 180,E1 -15757.746,E2 -15757.746} C_VEL
LIN {X 0,Y 312.667,Z 342.535,A -85,B 0,C 180,E1 -15761.672,E2 -15761.672} C_VEL
LIN {X 0,Y 312.698,Z 342.532,A -85,B 0,C 180,E1 -15764.888,E2 -15764.888} C_VEL
LIN {X 0,Y 312.628,Z 342.539,A -85,B 0,C 180,E1 -15769.237,E2 -15769.237} C_VEL
LIN {X 0,Y 312.544,Z 342.551,A -85,B 0,C 180,E1 -15772.79,E2 -15772.79} C_VEL
LIN {X 0,Y 312.601,Z 342.546,A -85,B 0,C 180,E1 -15775.936,E2 -15775.936} C_VEL
LIN {X 0,Y 312.536,Z 342.552,A -85,B 0,C 180,E1 -15779.651,E2 -15779.651} C_VEL
LIN {X 0,Y 312.518,Z 342.555,A -85,B 0,C 180,E1 -15783.69,E2 -15783.69} C_VEL
LIN {X 0,Y 312.536,Z 342.551,A -85,B 0,C 180,E1 -15787.384,E2 -15787.384} C_VEL
LIN {X 0,Y 312.489,Z 342.557,A -85,B 0,C 180,E1 -15790.71,E2 -15790.71} C_VEL
LIN {X 0,Y 312.451,Z 342.566,A -85,B 0,C 180,E1 -15794.21,E2 -15794.21} C_VEL
LIN {X 0,Y 312.484,Z 342.562,A -85,B 0,C 180,E1 -15797.919,E2 -15797.919} C_VEL
LIN {X 0,Y 312.535,Z 342.556,A -85,B 0,C 180,E1 -15801.911,E2 -15801.911} C_VEL
LIN {X 0,Y 312.507,Z 342.559,A -85,B 0,C 180,E1 -15805.791,E2 -15805.791} C_VEL
LIN {X 0,Y 312.603,Z 342.546,A -85,B 0,C 180,E1 -15809.647,E2 -15809.647} C_VEL
LIN {X 0,Y 319.511,Z 363.807,A -85,B 0,C 180,E1 -15810.66,E2 -15810.66} C_VEL
LIN {X 0,Y 317.848,Z 424.354,A -85,B 0,C 180,E1 -15812.465,E2 -15812.465} C_VEL
LIN {X 0,Y 317.114,Z 430.135,A -85,B 0,C 180,E1 -15812.649,E2 -15812.649} C_VEL
LIN {X 0,Y 314.131,Z 439.418,A -85,B 0,C 180,E1 -15812.985,E2 -15812.985} C_VEL
LIN {X 0,Y 310.997,Z 448.499,A -85,B 0,C 180,E1 -15813.448,E2 -15813.448} C_VEL
LIN {X 0,Y 310.034,Z 453.965,A -85,B 0,C 180,E1 -15813.829,E2 -15813.829} C_VEL
LIN {X 0,Y 309.338,Z 467.541,A -85,B 0,C 180,E1 -15815.034,E2 -15815.034} C_VEL
LIN {X 0,Y 308.576,Z 478.916,A -85,B 0,C 180,E1 -15816.334,E2 -15816.334} C_VEL
LIN {X 0,Y 307.76,Z 489.788,A -85,B 0,C 180,E1 -15817.865,E2 -15817.865} C_VEL
LIN {X 0,Y 306.985,Z 499.728,A -85,B 0,C 180,E1 -15819.602,E2 -15819.602} C_VEL
LIN {X 0,Y 306.292,Z 509.056,A -85,B 0,C 180,E1 -15821.61,E2 -15821.61} C_VEL
LIN {X 0,Y 305.698,Z 516.564,A -85,B 0,C 180,E1 -15823.643,E2 -15823.643} C_VEL
LIN {X 0,Y 305.422,Z 521.662,A -85,B 0,C 180,E1 -15825.339,E2 -15825.339} C_VEL
LIN {X 0,Y 305.168,Z 526.541,A -85,B 0,C 180,E1 -15827.363,E2 -15827.363} C_VEL
LIN {X 0,Y 305.106,Z 530.218,A -85,B 0,C 180,E1 -15829.382,E2 -15829.382} C_VEL
LIN {X 0,Y 305.179,Z 532.077,A -85,B 0,C 180,E1 -15830.724,E2 -15830.724} C_VEL
LIN {X 0,Y 305.31,Z 533.433,A -85,B 0,C 180,E1 -15832.062,E2 -15832.062} C_VEL
LIN {X 0,Y 305.466,Z 534.381,A -85,B 0,C 180,E1 -15833.395,E2 -15833.395} C_VEL
LIN {X 0,Y 305.593,Z 534.921,A -85,B 0,C 180,E1 -15834.722,E2 -15834.722} C_VEL
LIN {X 0,Y 305.949,Z 534.964,A -85,B 0,C 180,E1 -15836.049,E2 -15836.049} C_VEL
LIN {X 0,Y 306.383,Z 534.6,A -85,B 0,C 180,E1 -15837.371,E2 -15837.371} C_VEL
LIN {X 0,Y 306.885,Z 533.822,A -85,B 0,C 180,E1 -15838.688,E2 -15838.688} C_VEL
LIN {X 0,Y 307.463,Z 532.564,A -85,B 0,C 180,E1 -15840.001,E2 -15840.001} C_VEL
LIN {X 0,Y 308.56,Z 529.88,A -85,B 0,C 180,E1 -15841.959,E2 -15841.959} C_VEL
LIN {X 0,Y 310.008,Z 525.792,A -85,B 0,C 180,E1 -15844.047,E2 -15844.047} C_VEL
LIN {X 0,Y 311.564,Z 520.654,A -85,B 0,C 180,E1 -15846.018,E2 -15846.018} C_VEL
LIN {X 0,Y 313.48,Z 513.721,A -85,B 0,C 180,E1 -15848.055,E2 -15848.055} C_VEL
LIN {X 0,Y 315.511,Z 505.647,A -85,B 0,C 180,E1 -15849.941,E2 -15849.941} C_VEL
LIN {X 0,Y 317.321,Z 497.409,A -85,B 0,C 180,E1 -15851.498,E2 -15851.498} C_VEL
LIN {X 0,Y 319.477,Z 486.123,A -85,B 0,C 180,E1 -15853.194,E2 -15853.194} C_VEL
LIN {X 0,Y 321.148,Z 475.88,A -85,B 0,C 180,E1 -15854.415,E2 -15854.415} C_VEL
LIN {X 0,Y 322.732,Z 464.206,A -85,B 0,C 180,E1 -15855.533,E2 -15855.533} C_VEL
LIN {X 0,Y 323.956,Z 451.491,A -85,B 0,C 180,E1 -15856.483,E2 -15856.483} C_VEL
LIN {X 0,Y 324.821,Z 438.177,A -85,B 0,C 180,E1 -15857.201,E2 -15857.201} C_VEL
LIN {X 0,Y 326.512,Z 409.955,A -85,B 0,C 180,E1 -15858.248,E2 -15858.248} C_VEL
LIN {X 0,Y 328.869,Z 380.804,A -85,B 0,C 180,E1 -15859.283,E2 -15859.283} C_VEL
LIN {X 0,Y 323.948,Z 371.474,A -85,B 0,C 180,E1 -15860.684,E2 -15860.684} C_VEL
LIN {X 0,Y 318.319,Z 362.27,A -85,B 0,C 180,E1 -15862.425,E2 -15862.425} C_VEL
LIN {X 0,Y 315.358,Z 357.871,A -85,B 0,C 180,E1 -15863.425,E2 -15863.425} C_VEL
LIN {X 0,Y 313.154,Z 354.588,A -85,B 0,C 180,E1 -15864.22,E2 -15864.22} C_VEL
LIN {X 0,Y 312.155,Z 353.297,A -85,B 0,C 180,E1 -15864.594,E2 -15864.594} C_VEL
LIN {X 0,Y 310.168,Z 350.794,A -85,B 0,C 180,E1 -15865.357,E2 -15865.357} C_VEL
LIN {X 0,Y 309.105,Z 348.76,A -85,B 0,C 180,E1 -15865.838,E2 -15865.838} C_VEL
LIN {X 0,Y 306.779,Z 346.788,A -85,B 0,C 180,E1 -15866.773,E2 -15866.773} C_VEL
LIN {X 0,Y 305.563,Z 344.154,A -85,B 0,C 180,E1 -15867.434,E2 -15867.434} C_VEL
LIN {X 0,Y 305.449,Z 343.437,A -85,B 0,C 180,E1 -15867.585,E2 -15867.585} C_VEL
LIN {X 0,Y 305.44,Z 343.437,A -85,B 0,C 180,E1 -15871.953,E2 -15871.953} C_VEL
LIN {X 0,Y 305.465,Z 343.43,A -85,B 0,C 180,E1 -15875.114,E2 -15875.114} C_VEL
LIN {X 0,Y 305.419,Z 343.436,A -85,B 0,C 180,E1 -15878.521,E2 -15878.521} C_VEL
LIN {X 0,Y 305.438,Z 343.434,A -85,B 0,C 180,E1 -15882.582,E2 -15882.582} C_VEL
LIN {X 0,Y 305.425,Z 343.441,A -85,B 0,C 180,E1 -15886.344,E2 -15886.344} C_VEL
LIN {X 0,Y 305.443,Z 343.631,A -85,B 0,C 180,E1 -15890.191,E2 -15890.191} C_VEL
LIN {X 0,Y 306.516,Z 346.4,A -85,B 0,C 180,E1 -15891.223,E2 -15891.223} C_VEL
LIN {X 0,Y 308.744,Z 348.908,A -85,B 0,C 180,E1 -15892.506,E2 -15892.506} C_VEL
LIN {X 0,Y 310.3,Z 351.944,A -85,B 0,C 180,E1 -15893.52,E2 -15893.52} C_VEL
LIN {X 0,Y 311.731,Z 353.872,A -85,B 0,C 180,E1 -15894.256,E2 -15894.256} C_VEL
LIN {X 0,Y 315.647,Z 369.108,A -85,B 0,C 180,E1 -15897.18,E2 -15897.18} C_VEL
LIN {X 0,Y 318.753,Z 378.979,A -85,B 0,C 180,E1 -15898.509,E2 -15898.509} C_VEL
LIN {X 0,Y 320.673,Z 394.734,A -85,B 0,C 180,E1 -15899.796,E2 -15899.796} C_VEL
LIN {X 0,Y 322.525,Z 414.155,A -85,B 0,C 180,E1 -15901.161,E2 -15901.161} C_VEL
LIN {X 0,Y 323.881,Z 433.847,A -85,B 0,C 180,E1 -15902.362,E2 -15902.362} C_VEL
LIN {X 0,Y 324.402,Z 453.744,A -85,B 0,C 180,E1 -15903.386,E2 -15903.386} C_VEL
LIN {X 0,Y 321.162,Z 498.548,A -85,B 0,C 180,E1 -15904.957,E2 -15904.957} C_VEL
LIN {X 0,Y 319.634,Z 512.076,A -85,B 0,C 180,E1 -15905.652,E2 -15905.652} C_VEL
LIN {X 0,Y 317.548,Z 524.811,A -85,B 0,C 180,E1 -15906.523,E2 -15906.523} C_VEL
LIN {X 0,Y 315.135,Z 538.161,A -85,B 0,C 180,E1 -15907.72,E2 -15907.72} C_VEL
LIN {X 0,Y 312.735,Z 550.021,A -85,B 0,C 180,E1 -15909.099,E2 -15909.099} C_VEL
LIN {X 0,Y 310.798,Z 559.793,A -85,B 0,C 180,E1 -15910.516,E2 -15910.516} C_VEL
LIN {X 0,Y 308.752,Z 568.924,A -85,B 0,C 180,E1 -15912.103,E2 -15912.103} C_VEL
LIN {X 0,Y 306.864,Z 578.309,A -85,B 0,C 180,E1 -15914.138,E2 -15914.138} C_VEL
LIN {X 0,Y 305.632,Z 585.361,A -85,B 0,C 180,E1 -15916.028,E2 -15916.028} C_VEL
LIN {X 0,Y 304.782,Z 591.416,A -85,B 0,C 180,E1 -15918.022,E2 -15918.022} C_VEL
LIN {X 0,Y 304.297,Z 596.258,A -85,B 0,C 180,E1 -15920.025,E2 -15920.025} C_VEL
LIN {X 0,Y 304.149,Z 599.983,A -85,B 0,C 180,E1 -15922.03,E2 -15922.03} C_VEL
LIN {X 0,Y 304.283,Z 601.893,A -85,B 0,C 180,E1 -15923.368,E2 -15923.368} C_VEL
LIN {X 0,Y 304.393,Z 603.339,A -85,B 0,C 180,E1 -15924.701,E2 -15924.701} C_VEL
LIN {X 0,Y 304.629,Z 604.368,A -85,B 0,C 180,E1 -15926.031,E2 -15926.031} C_VEL
LIN {X 0,Y 304.801,Z 604.941,A -85,B 0,C 180,E1 -15927.357,E2 -15927.357} C_VEL
LIN {X 0,Y 304.985,Z 605.023,A -85,B 0,C 180,E1 -15928.679,E2 -15928.679} C_VEL
LIN {X 0,Y 305.061,Z 605.746,A -85,B 0,C 180,E1 -15930,E2 -15930} C_VEL
LIN {X 0,Y 304.849,Z 606.185,A -85,B 0,C 180,E1 -15931.321,E2 -15931.321} C_VEL
LIN {X 0,Y 304.705,Z 606.185,A -85,B 0,C 180,E1 -15932.644,E2 -15932.644} C_VEL
LIN {X 0,Y 304.545,Z 605.739,A -85,B 0,C 180,E1 -15933.97,E2 -15933.97} C_VEL
LIN {X 0,Y 304.298,Z 604.823,A -85,B 0,C 180,E1 -15935.301,E2 -15935.301} C_VEL
LIN {X 0,Y 304.2,Z 603.453,A -85,B 0,C 180,E1 -15936.633,E2 -15936.633} C_VEL
LIN {X 0,Y 304.118,Z 600.586,A -85,B 0,C 180,E1 -15938.639,E2 -15938.639} C_VEL
LIN {X 0,Y 304.322,Z 596.696,A -85,B 0,C 180,E1 -15940.646,E2 -15940.646} C_VEL
LIN {X 0,Y 305.031,Z 591.727,A -85,B 0,C 180,E1 -15942.643,E2 -15942.643} C_VEL
LIN {X 0,Y 306.114,Z 585.555,A -85,B 0,C 180,E1 -15944.628,E2 -15944.628} C_VEL
LIN {X 0,Y 307.58,Z 578.044,A -85,B 0,C 180,E1 -15946.596,E2 -15946.596} C_VEL
LIN {X 0,Y 309.588,Z 568.956,A -85,B 0,C 180,E1 -15948.531,E2 -15948.531} C_VEL
LIN {X 0,Y 311.982,Z 558.827,A -85,B 0,C 180,E1 -15950.264,E2 -15950.264} C_VEL
LIN {X 0,Y 314.474,Z 547.731,A -85,B 0,C 180,E1 -15951.811,E2 -15951.811} C_VEL
LIN {X 0,Y 317.118,Z 535.567,A -85,B 0,C 180,E1 -15953.165,E2 -15953.165} C_VEL
